//     Term 1 (AT2202-0500)/CC Inputs/Current actual value Ch.9 <-> Data Pointer/CurrentActualValues[8]
//     Term 1 (AT2202-0500)/CC Inputs/Status <-> Data Pointer/Status
//     Term 1 (AT2202-0500)/CC Outputs/Control <-> Data Pointer/Control
//     Term 1 (AT2202-0500)/CC Outputs/Current setpoint value Ch.1 <-> Data Pointer/CurrentSetpointValues[0]
//     Term 1 (AT2202-0500)/CC Outputs/Current setpoint value Ch.10 <-> Data Pointer/CurrentSetpointValues[9]
//     Term 1 (AT2202-0500)/CC Outputs/Current setpoint value Ch.11 <-> Data Pointer/CurrentSetpointValues[10]
//     Term 1 (AT2202-0500)/CC Outputs/Current setpoint value Ch.12 <-> Data Pointer/CurrentSetpointValues[11]
//     Term 1 (AT2202-0500)/CC Outputs/Current setpoint value Ch.13 <-> Data Pointer/CurrentSetpointValues[12]
//     Term 1 (AT2202-0500)/CC Outputs/Current setpoint value Ch.14 <-> Data Pointer/CurrentSetpointValues[13]
//     Term 1 (AT2202-0500)/CC Outputs/Current setpoint value Ch.15 <-> Data Pointer/CurrentSetpointValues[14]
//     Term 1 (AT2202-0500)/CC Outputs/Current setpoint value Ch.16 <-> Data Pointer/CurrentSetpointValues[15]
//     Term 1 (AT2202-0500)/CC Outputs/Current setpoint value Ch.17 <-> Data Pointer/CurrentSetpointValues[16]
//     Term 1 (AT2202-0500)/CC Outputs/Current setpoint value Ch.18 <-> Data Pointer/CurrentSetpointValues[17]
//     Term 1 (AT2202-0500)/CC Outputs/Current setpoint value Ch.19 <-> Data Pointer/CurrentSetpointValues[18]
//     Term 1 (AT2202-0500)/CC Outputs/Current setpoint value Ch.2 <-> Data Pointer/CurrentSetpointValues[1]
//     Term 1 (AT2202-0500)/CC Outputs/Current setpoint value Ch.20 <-> Data Pointer/CurrentSetpointValues[19]
//     Term 1 (AT2202-0500)/CC Outputs/Current setpoint value Ch.21 <-> Data Pointer/CurrentSetpointValues[20]
//     Term 1 (AT2202-0500)/CC Outputs/Current setpoint value Ch.22 <-> Data Pointer/CurrentSetpointValues[21]
//     Term 1 (AT2202-0500)/CC Outputs/Current setpoint value Ch.23 <-> Data Pointer/CurrentSetpointValues[22]
//     Term 1 (AT2202-0500)/CC Outputs/Current setpoint value Ch.24 <-> Data Pointer/CurrentSetpointValues[23]
//     Term 1 (AT2202-0500)/CC Outputs/Current setpoint value Ch.25 <-> Data Pointer/CurrentSetpointValues[24]
//     Term 1 (AT2202-0500)/CC Outputs/Current setpoint value Ch.26 <-> Data Pointer/CurrentSetpointValues[25]
//     Term 1 (AT2202-0500)/CC Outputs/Current setpoint value Ch.27 <-> Data Pointer/CurrentSetpointValues[26]
//     Term 1 (AT2202-0500)/CC Outputs/Current setpoint value Ch.28 <-> Data Pointer/CurrentSetpointValues[27]
//     Term 1 (AT2202-0500)/CC Outputs/Current setpoint value Ch.29 <-> Data Pointer/CurrentSetpointValues[28]
//     Term 1 (AT2202-0500)/CC Outputs/Current setpoint value Ch.3 <-> Data Pointer/CurrentSetpointValues[2]
//     Term 1 (AT2202-0500)/CC Outputs/Current setpoint value Ch.30 <-> Data Pointer/CurrentSetpointValues[29]
//     Term 1 (AT2202-0500)/CC Outputs/Current setpoint value Ch.4 <-> Data Pointer/CurrentSetpointValues[3]
//     Term 1 (AT2202-0500)/CC Outputs/Current setpoint value Ch.5 <-> Data Pointer/CurrentSetpointValues[4]
//     Term 1 (AT2202-0500)/CC Outputs/Current setpoint value Ch.6 <-> Data Pointer/CurrentSetpointValues[5]
//     Term 1 (AT2202-0500)/CC Outputs/Current setpoint value Ch.7 <-> Data Pointer/CurrentSetpointValues[6]
//     Term 1 (AT2202-0500)/CC Outputs/Current setpoint value Ch.8 <-> Data Pointer/CurrentSetpointValues[7]
//     Term 1 (AT2202-0500)/CC Outputs/Current setpoint value Ch.9 <-> Data Pointer/CurrentSetpointValues[8]
//     Term 1 (AT2202-0500)/LFB Inputs/BinaryData <-> Data Pointer/HallSensorValues
//   Device 1 <-> TcCOM Objects/XTS ProcessingUnit 1/Part 1/Module 2
//     Term 2 (AT2200-0500)/CC Inputs/Current actual value Ch.1 <-> Data Pointer/CurrentActualValues[0]
//     Term 2 (AT2200-0500)/CC Inputs/Current actual value Ch.10 <-> Data Pointer/CurrentActualValues[9]
//     Term 2 (AT2200-0500)/CC Inputs/Current actual value Ch.11 <-> Data Pointer/CurrentActualValues[10]
//     Term 2 (AT2200-0500)/CC Inputs/Current actual value Ch.12 <-> Data Pointer/CurrentActualValues[11]
//     Term 2 (AT2200-0500)/CC Inputs/Current actual value Ch.13 <-> Data Pointer/CurrentActualValues[12]
//     Term 2 (AT2200-0500)/CC Inputs/Current actual value Ch.14 <-> Data Pointer/CurrentActualValues[13]
//     Term 2 (AT2200-0500)/CC Inputs/Current actual value Ch.15 <-> Data Pointer/CurrentActualValues[14]
//     Term 2 (AT2200-0500)/CC Inputs/Current actual value Ch.16 <-> Data Pointer/CurrentActualValues[15]
//     Term 2 (AT2200-0500)/CC Inputs/Current actual value Ch.17 <-> Data Pointer/CurrentActualValues[16]
//     Term 2 (AT2200-0500)/CC Inputs/Current actual value Ch.18 <-> Data Pointer/CurrentActualValues[17]
//     Term 2 (AT2200-0500)/CC Inputs/Current actual value Ch.19 <-> Data Pointer/CurrentActualValues[18]
//     Term 2 (AT2200-0500)/CC Inputs/Current actual value Ch.2 <-> Data Pointer/CurrentActualValues[1]
//     Term 2 (AT2200-0500)/CC Inputs/Current actual value Ch.20 <-> Data Pointer/CurrentActualValues[19]
//     Term 2 (AT2200-0500)/CC Inputs/Current actual value Ch.21 <-> Data Pointer/CurrentActualValues[20]
//     Term 2 (AT2200-0500)/CC Inputs/Current actual value Ch.22 <-> Data Pointer/CurrentActualValues[21]
//     Term 2 (AT2200-0500)/CC Inputs/Current actual value Ch.23 <-> Data Pointer/CurrentActualValues[22]
//     Term 2 (AT2200-0500)/CC Inputs/Current actual value Ch.24 <-> Data Pointer/CurrentActualValues[23]
//     Term 2 (AT2200-0500)/CC Inputs/Current actual value Ch.25 <-> Data Pointer/CurrentActualValues[24]
//     Term 2 (AT2200-0500)/CC Inputs/Current actual value Ch.26 <-> Data Pointer/CurrentActualValues[25]
//     Term 2 (AT2200-0500)/CC Inputs/Current actual value Ch.27 <-> Data Pointer/CurrentActualValues[26]
//     Term 2 (AT2200-0500)/CC Inputs/Current actual value Ch.28 <-> Data Pointer/CurrentActualValues[27]
//     Term 2 (AT2200-0500)/CC Inputs/Current actual value Ch.29 <-> Data Pointer/CurrentActualValues[28]
//     Term 2 (AT2200-0500)/CC Inputs/Current actual value Ch.3 <-> Data Pointer/CurrentActualValues[2]
//     Term 2 (AT2200-0500)/CC Inputs/Current actual value Ch.30 <-> Data Pointer/CurrentActualValues[29]
//     Term 2 (AT2200-0500)/CC Inputs/Current actual value Ch.4 <-> Data Pointer/CurrentActualValues[3]
//     Term 2 (AT2200-0500)/CC Inputs/Current actual value Ch.5 <-> Data Pointer/CurrentActualValues[4]
//     Term 2 (AT2200-0500)/CC Inputs/Current actual value Ch.6 <-> Data Pointer/CurrentActualValues[5]
//     Term 2 (AT2200-0500)/CC Inputs/Current actual value Ch.7 <-> Data Pointer/CurrentActualValues[6]
//     Term 2 (AT2200-0500)/CC Inputs/Current actual value Ch.8 <-> Data Pointer/CurrentActualValues[7]
//     Term 2 (AT2200-0500)/CC Inputs/Current actual value Ch.9 <-> Data Pointer/CurrentActualValues[8]
//     Term 2 (AT2200-0500)/CC Inputs/Status <-> Data Pointer/Status
//     Term 2 (AT2200-0500)/CC Outputs/Control <-> Data Pointer/Control
//     Term 2 (AT2200-0500)/CC Outputs/Current setpoint value Ch.1 <-> Data Pointer/CurrentSetpointValues[0]
//     Term 2 (AT2200-0500)/CC Outputs/Current setpoint value Ch.10 <-> Data Pointer/CurrentSetpointValues[9]
//     Term 2 (AT2200-0500)/CC Outputs/Current setpoint value Ch.11 <-> Data Pointer/CurrentSetpointValues[10]
//     Term 2 (AT2200-0500)/CC Outputs/Current setpoint value Ch.12 <-> Data Pointer/CurrentSetpointValues[11]
//     Term 2 (AT2200-0500)/CC Outputs/Current setpoint value Ch.13 <-> Data Pointer/CurrentSetpointValues[12]
//     Term 2 (AT2200-0500)/CC Outputs/Current setpoint value Ch.14 <-> Data Pointer/CurrentSetpointValues[13]
//     Term 2 (AT2200-0500)/CC Outputs/Current setpoint value Ch.15 <-> Data Pointer/CurrentSetpointValues[14]
//     Term 2 (AT2200-0500)/CC Outputs/Current setpoint value Ch.16 <-> Data Pointer/CurrentSetpointValues[15]
//     Term 2 (AT2200-0500)/CC Outputs/Current setpoint value Ch.17 <-> Data Pointer/CurrentSetpointValues[16]
//     Term 2 (AT2200-0500)/CC Outputs/Current setpoint value Ch.18 <-> Data Pointer/CurrentSetpointValues[17]
//     Term 2 (AT2200-0500)/CC Outputs/Current setpoint value Ch.19 <-> Data Pointer/CurrentSetpointValues[18]
//     Term 2 (AT2200-0500)/CC Outputs/Current setpoint value Ch.2 <-> Data Pointer/CurrentSetpointValues[1]
//     Term 2 (AT2200-0500)/CC Outputs/Current setpoint value Ch.20 <-> Data Pointer/CurrentSetpointValues[19]
//     Term 2 (AT2200-0500)/CC Outputs/Current setpoint value Ch.21 <-> Data Pointer/CurrentSetpointValues[20]
//     Term 2 (AT2200-0500)/CC Outputs/Current setpoint value Ch.22 <-> Data Pointer/CurrentSetpointValues[21]
//     Term 2 (AT2200-0500)/CC Outputs/Current setpoint value Ch.23 <-> Data Pointer/CurrentSetpointValues[22]
//     Term 2 (AT2200-0500)/CC Outputs/Current setpoint value Ch.24 <-> Data Pointer/CurrentSetpointValues[23]
//     Term 2 (AT2200-0500)/CC Outputs/Current setpoint value Ch.25 <-> Data Pointer/CurrentSetpointValues[24]
//     Term 2 (AT2200-0500)/CC Outputs/Current setpoint value Ch.26 <-> Data Pointer/CurrentSetpointValues[25]
//     Term 2 (AT2200-0500)/CC Outputs/Current setpoint value Ch.27 <-> Data Pointer/CurrentSetpointValues[26]
//     Term 2 (AT2200-0500)/CC Outputs/Current setpoint value Ch.28 <-> Data Pointer/CurrentSetpointValues[27]
//     Term 2 (AT2200-0500)/CC Outputs/Current setpoint value Ch.29 <-> Data Pointer/CurrentSetpointValues[28]
//     Term 2 (AT2200-0500)/CC Outputs/Current setpoint value Ch.3 <-> Data Pointer/CurrentSetpointValues[2]
//     Term 2 (AT2200-0500)/CC Outputs/Current setpoint value Ch.30 <-> Data Pointer/CurrentSetpointValues[29]
//     Term 2 (AT2200-0500)/CC Outputs/Current setpoint value Ch.4 <-> Data Pointer/CurrentSetpointValues[3]
//     Term 2 (AT2200-0500)/CC Outputs/Current setpoint value Ch.5 <-> Data Pointer/CurrentSetpointValues[4]
//     Term 2 (AT2200-0500)/CC Outputs/Current setpoint value Ch.6 <-> Data Pointer/CurrentSetpointValues[5]
//     Term 2 (AT2200-0500)/CC Outputs/Current setpoint value Ch.7 <-> Data Pointer/CurrentSetpointValues[6]
//     Term 2 (AT2200-0500)/CC Outputs/Current setpoint value Ch.8 <-> Data Pointer/CurrentSetpointValues[7]
//     Term 2 (AT2200-0500)/CC Outputs/Current setpoint value Ch.9 <-> Data Pointer/CurrentSetpointValues[8]
//     Term 2 (AT2200-0500)/LFB Inputs/BinaryData <-> Data Pointer/HallSensorValues
//   Device 1 <-> TcCOM Objects/XTS ProcessingUnit 1/Part 1/Module 3
//     Term 3 (AT2200-0500)/CC Inputs/Current actual value Ch.1 <-> Data Pointer/CurrentActualValues[0]
//     Term 3 (AT2200-0500)/CC Inputs/Current actual value Ch.10 <-> Data Pointer/CurrentActualValues[9]
//     Term 3 (AT2200-0500)/CC Inputs/Current actual value Ch.11 <-> Data Pointer/CurrentActualValues[10]
//     Term 3 (AT2200-0500)/CC Inputs/Current actual value Ch.12 <-> Data Pointer/CurrentActualValues[11]
//     Term 3 (AT2200-0500)/CC Inputs/Current actual value Ch.13 <-> Data Pointer/CurrentActualValues[12]
//     Term 3 (AT2200-0500)/CC Inputs/Current actual value Ch.14 <-> Data Pointer/CurrentActualValues[13]
//     Term 3 (AT2200-0500)/CC Inputs/Current actual value Ch.15 <-> Data Pointer/CurrentActualValues[14]
//     Term 3 (AT2200-0500)/CC Inputs/Current actual value Ch.16 <-> Data Pointer/CurrentActualValues[15]
//     Term 3 (AT2200-0500)/CC Inputs/Current actual value Ch.17 <-> Data Pointer/CurrentActualValues[16]
//     Term 3 (AT2200-0500)/CC Inputs/Current actual value Ch.18 <-> Data Pointer/CurrentActualValues[17]
//     Term 3 (AT2200-0500)/CC Inputs/Current actual value Ch.19 <-> Data Pointer/CurrentActualValues[18]
//     Term 3 (AT2200-0500)/CC Inputs/Current actual value Ch.2 <-> Data Pointer/CurrentActualValues[1]
//     Term 3 (AT2200-0500)/CC Inputs/Current actual value Ch.20 <-> Data Pointer/CurrentActualValues[19]
//     Term 3 (AT2200-0500)/CC Inputs/Current actual value Ch.21 <-> Data Pointer/CurrentActualValues[20]
//     Term 3 (AT2200-0500)/CC Inputs/Current actual value Ch.22 <-> Data Pointer/CurrentActualValues[21]
//     Term 3 (AT2200-0500)/CC Inputs/Current actual value Ch.23 <-> Data Pointer/CurrentActualValues[22]
//     Term 3 (AT2200-0500)/CC Inputs/Current actual value Ch.24 <-> Data Pointer/CurrentActualValues[23]
//     Term 3 (AT2200-0500)/CC Inputs/Current actual value Ch.25 <-> Data Pointer/CurrentActualValues[24]
//     Term 3 (AT2200-0500)/CC Inputs/Current actual value Ch.26 <-> Data Pointer/CurrentActualValues[25]
//     Term 3 (AT2200-0500)/CC Inputs/Current actual value Ch.27 <-> Data Pointer/CurrentActualValues[26]
//     Term 3 (AT2200-0500)/CC Inputs/Current actual value Ch.28 <-> Data Pointer/CurrentActualValues[27]
//     Term 3 (AT2200-0500)/CC Inputs/Current actual value Ch.29 <-> Data Pointer/CurrentActualValues[28]
//     Term 3 (AT2200-0500)/CC Inputs/Current actual value Ch.3 <-> Data Pointer/CurrentActualValues[2]
//     Term 3 (AT2200-0500)/CC Inputs/Current actual value Ch.30 <-> Data Pointer/CurrentActualValues[29]
//     Term 3 (AT2200-0500)/CC Inputs/Current actual value Ch.4 <-> Data Pointer/CurrentActualValues[3]
//     Term 3 (AT2200-0500)/CC Inputs/Current actual value Ch.5 <-> Data Pointer/CurrentActualValues[4]
//     Term 3 (AT2200-0500)/CC Inputs/Current actual value Ch.6 <-> Data Pointer/CurrentActualValues[5]
//     Term 3 (AT2200-0500)/CC Inputs/Current actual value Ch.7 <-> Data Pointer/CurrentActualValues[6]
//     Term 3 (AT2200-0500)/CC Inputs/Current actual value Ch.8 <-> Data Pointer/CurrentActualValues[7]
//     Term 3 (AT2200-0500)/CC Inputs/Current actual value Ch.9 <-> Data Pointer/CurrentActualValues[8]
//     Term 3 (AT2200-0500)/CC Inputs/Status <-> Data Pointer/Status
//     Term 3 (AT2200-0500)/CC Outputs/Control <-> Data Pointer/Control
//     Term 3 (AT2200-0500)/CC Outputs/Current setpoint value Ch.1 <-> Data Pointer/CurrentSetpointValues[0]
//     Term 3 (AT2200-0500)/CC Outputs/Current setpoint value Ch.10 <-> Data Pointer/CurrentSetpointValues[9]
//     Term 3 (AT2200-0500)/CC Outputs/Current setpoint value Ch.11 <-> Data Pointer/CurrentSetpointValues[10]
//     Term 3 (AT2200-0500)/CC Outputs/Current setpoint value Ch.12 <-> Data Pointer/CurrentSetpointValues[11]
//     Term 3 (AT2200-0500)/CC Outputs/Current setpoint value Ch.13 <-> Data Pointer/CurrentSetpointValues[12]
//     Term 3 (AT2200-0500)/CC Outputs/Current setpoint value Ch.14 <-> Data Pointer/CurrentSetpointValues[13]
//     Term 3 (AT2200-0500)/CC Outputs/Current setpoint value Ch.15 <-> Data Pointer/CurrentSetpointValues[14]
//     Term 3 (AT2200-0500)/CC Outputs/Current setpoint value Ch.16 <-> Data Pointer/CurrentSetpointValues[15]
//     Term 3 (AT2200-0500)/CC Outputs/Current setpoint value Ch.17 <-> Data Pointer/CurrentSetpointValues[16]
//     Term 3 (AT2200-0500)/CC Outputs/Current setpoint value Ch.18 <-> Data Pointer/CurrentSetpointValues[17]
//     Term 3 (AT2200-0500)/CC Outputs/Current setpoint value Ch.19 <-> Data Pointer/CurrentSetpointValues[18]
//     Term 3 (AT2200-0500)/CC Outputs/Current setpoint value Ch.2 <-> Data Pointer/CurrentSetpointValues[1]
//     Term 3 (AT2200-0500)/CC Outputs/Current setpoint value Ch.20 <-> Data Pointer/CurrentSetpointValues[19]
//     Term 3 (AT2200-0500)/CC Outputs/Current setpoint value Ch.21 <-> Data Pointer/CurrentSetpointValues[20]
//     Term 3 (AT2200-0500)/CC Outputs/Current setpoint value Ch.22 <-> Data Pointer/CurrentSetpointValues[21]
//     Term 3 (AT2200-0500)/CC Outputs/Current setpoint value Ch.23 <-> Data Pointer/CurrentSetpointValues[22]
//     Term 3 (AT2200-0500)/CC Outputs/Current setpoint value Ch.24 <-> Data Pointer/CurrentSetpointValues[23]
//     Term 3 (AT2200-0500)/CC Outputs/Current setpoint value Ch.25 <-> Data Pointer/CurrentSetpointValues[24]
//     Term 3 (AT2200-0500)/CC Outputs/Current setpoint value Ch.26 <-> Data Pointer/CurrentSetpointValues[25]
//     Term 3 (AT2200-0500)/CC Outputs/Current setpoint value Ch.27 <-> Data Pointer/CurrentSetpointValues[26]
//     Term 3 (AT2200-0500)/CC Outputs/Current setpoint value Ch.28 <-> Data Pointer/CurrentSetpointValues[27]
//     Term 3 (AT2200-0500)/CC Outputs/Current setpoint value Ch.29 <-> Data Pointer/CurrentSetpointValues[28]
//     Term 3 (AT2200-0500)/CC Outputs/Current setpoint value Ch.3 <-> Data Pointer/CurrentSetpointValues[2]
//     Term 3 (AT2200-0500)/CC Outputs/Current setpoint value Ch.30 <-> Data Pointer/CurrentSetpointValues[29]
//     Term 3 (AT2200-0500)/CC Outputs/Current setpoint value Ch.4 <-> Data Pointer/CurrentSetpointValues[3]
//     Term 3 (AT2200-0500)/CC Outputs/Current setpoint value Ch.5 <-> Data Pointer/CurrentSetpointValues[4]
//     Term 3 (AT2200-0500)/CC Outputs/Current setpoint value Ch.6 <-> Data Pointer/CurrentSetpointValues[5]
//     Term 3 (AT2200-0500)/CC Outputs/Current setpoint value Ch.7 <-> Data Pointer/CurrentSetpointValues[6]
//     Term 3 (AT2200-0500)/CC Outputs/Current setpoint value Ch.8 <-> Data Pointer/CurrentSetpointValues[7]
//     Term 3 (AT2200-0500)/CC Outputs/Current setpoint value Ch.9 <-> Data Pointer/CurrentSetpointValues[8]
//     Term 3 (AT2200-0500)/LFB Inputs/BinaryData <-> Data Pointer/HallSensorValues
//   Device 16 <-> TcCOM Objects/XTS ProcessingUnit 1/Part 1/Module 4
//     Term 4 (AT2202-0500)/CC Inputs/Current actual value Ch.1 <-> Data Pointer/CurrentActualValues[0]
//     Term 4 (AT2202-0500)/CC Inputs/Current actual value Ch.10 <-> Data Pointer/CurrentActualValues[9]
//     Term 4 (AT2202-0500)/CC Inputs/Current actual value Ch.11 <-> Data Pointer/CurrentActualValues[10]
//     Term 4 (AT2202-0500)/CC Inputs/Current actual value Ch.12 <-> Data Pointer/CurrentActualValues[11]
//     Term 4 (AT2202-0500)/CC Inputs/Current actual value Ch.13 <-> Data Pointer/CurrentActualValues[12]
//     Term 4 (AT2202-0500)/CC Inputs/Current actual value Ch.14 <-> Data Pointer/CurrentActualValues[13]
//     Term 4 (AT2202-0500)/CC Inputs/Current actual value Ch.15 <-> Data Pointer/CurrentActualValues[14]
//     Term 4 (AT2202-0500)/CC Inputs/Current actual value Ch.16 <-> Data Pointer/CurrentActualValues[15]
//     Term 4 (AT2202-0500)/CC Inputs/Current actual value Ch.17 <-> Data Pointer/CurrentActualValues[16]
//     Term 4 (AT2202-0500)/CC Inputs/Current actual value Ch.18 <-> Data Pointer/CurrentActualValues[17]
//     Term 4 (AT2202-0500)/CC Inputs/Current actual value Ch.19 <-> Data Pointer/CurrentActualValues[18]
//     Term 4 (AT2202-0500)/CC Inputs/Current actual value Ch.2 <-> Data Pointer/CurrentActualValues[1]
//     Term 4 (AT2202-0500)/CC Inputs/Current actual value Ch.20 <-> Data Pointer/CurrentActualValues[19]
//     Term 4 (AT2202-0500)/CC Inputs/Current actual value Ch.21 <-> Data Pointer/CurrentActualValues[20]
//     Term 4 (AT2202-0500)/CC Inputs/Current actual value Ch.22 <-> Data Pointer/CurrentActualValues[21]
//     Term 4 (AT2202-0500)/CC Inputs/Current actual value Ch.23 <-> Data Pointer/CurrentActualValues[22]
//     Term 4 (AT2202-0500)/CC Inputs/Current actual value Ch.24 <-> Data Pointer/CurrentActualValues[23]
//     Term 4 (AT2202-0500)/CC Inputs/Current actual value Ch.25 <-> Data Pointer/CurrentActualValues[24]
//     Term 4 (AT2202-0500)/CC Inputs/Current actual value Ch.26 <-> Data Pointer/CurrentActualValues[25]
//     Term 4 (AT2202-0500)/CC Inputs/Current actual value Ch.27 <-> Data Pointer/CurrentActualValues[26]
//     Term 4 (AT2202-0500)/CC Inputs/Current actual value Ch.28 <-> Data Pointer/CurrentActualValues[27]
//     Term 4 (AT2202-0500)/CC Inputs/Current actual value Ch.29 <-> Data Pointer/CurrentActualValues[28]
//     Term 4 (AT2202-0500)/CC Inputs/Current actual value Ch.3 <-> Data Pointer/CurrentActualValues[2]
//     Term 4 (AT2202-0500)/CC Inputs/Current actual value Ch.30 <-> Data Pointer/CurrentActualValues[29]
//     Term 4 (AT2202-0500)/CC Inputs/Current actual value Ch.4 <-> Data Pointer/CurrentActualValues[3]
//     Term 4 (AT2202-0500)/CC Inputs/Current actual value Ch.5 <-> Data Pointer/CurrentActualValues[4]
//     Term 4 (AT2202-0500)/CC Inputs/Current actual value Ch.6 <-> Data Pointer/CurrentActualValues[5]
//     Term 4 (AT2202-0500)/CC Inputs/Current actual value Ch.7 <-> Data Pointer/CurrentActualValues[6]
//     Term 4 (AT2202-0500)/CC Inputs/Current actual value Ch.8 <-> Data Pointer/CurrentActualValues[7]
//     Term 4 (AT2202-0500)/CC Inputs/Current actual value Ch.9 <-> Data Pointer/CurrentActualValues[8]
//     Term 4 (AT2202-0500)/CC Inputs/Status <-> Data Pointer/Status
//     Term 4 (AT2202-0500)/CC Outputs/Control <-> Data Pointer/Control
//     Term 4 (AT2202-0500)/CC Outputs/Current setpoint value Ch.1 <-> Data Pointer/CurrentSetpointValues[0]
//     Term 4 (AT2202-0500)/CC Outputs/Current setpoint value Ch.10 <-> Data Pointer/CurrentSetpointValues[9]
//     Term 4 (AT2202-0500)/CC Outputs/Current setpoint value Ch.11 <-> Data Pointer/CurrentSetpointValues[10]
//     Term 4 (AT2202-0500)/CC Outputs/Current setpoint value Ch.12 <-> Data Pointer/CurrentSetpointValues[11]
//     Term 4 (AT2202-0500)/CC Outputs/Current setpoint value Ch.13 <-> Data Pointer/CurrentSetpointValues[12]
//     Term 4 (AT2202-0500)/CC Outputs/Current setpoint value Ch.14 <-> Data Pointer/CurrentSetpointValues[13]
//     Term 4 (AT2202-0500)/CC Outputs/Current setpoint value Ch.15 <-> Data Pointer/CurrentSetpointValues[14]
//     Term 4 (AT2202-0500)/CC Outputs/Current setpoint value Ch.16 <-> Data Pointer/CurrentSetpointValues[15]
//     Term 4 (AT2202-0500)/CC Outputs/Current setpoint value Ch.17 <-> Data Pointer/CurrentSetpointValues[16]
//     Term 4 (AT2202-0500)/CC Outputs/Current setpoint value Ch.18 <-> Data Pointer/CurrentSetpointValues[17]
//     Term 4 (AT2202-0500)/CC Outputs/Current setpoint value Ch.19 <-> Data Pointer/CurrentSetpointValues[18]
//     Term 4 (AT2202-0500)/CC Outputs/Current setpoint value Ch.2 <-> Data Pointer/CurrentSetpointValues[1]
//     Term 4 (AT2202-0500)/CC Outputs/Current setpoint value Ch.20 <-> Data Pointer/CurrentSetpointValues[19]
//     Term 4 (AT2202-0500)/CC Outputs/Current setpoint value Ch.21 <-> Data Pointer/CurrentSetpointValues[20]
//     Term 4 (AT2202-0500)/CC Outputs/Current setpoint value Ch.22 <-> Data Pointer/CurrentSetpointValues[21]
//     Term 4 (AT2202-0500)/CC Outputs/Current setpoint value Ch.23 <-> Data Pointer/CurrentSetpointValues[22]
//     Term 4 (AT2202-0500)/CC Outputs/Current setpoint value Ch.24 <-> Data Pointer/CurrentSetpointValues[23]
//     Term 4 (AT2202-0500)/CC Outputs/Current setpoint value Ch.25 <-> Data Pointer/CurrentSetpointValues[24]
//     Term 4 (AT2202-0500)/CC Outputs/Current setpoint value Ch.26 <-> Data Pointer/CurrentSetpointValues[25]
//     Term 4 (AT2202-0500)/CC Outputs/Current setpoint value Ch.27 <-> Data Pointer/CurrentSetpointValues[26]
//     Term 4 (AT2202-0500)/CC Outputs/Current setpoint value Ch.28 <-> Data Pointer/CurrentSetpointValues[27]
//     Term 4 (AT2202-0500)/CC Outputs/Current setpoint value Ch.29 <-> Data Pointer/CurrentSetpointValues[28]
//     Term 4 (AT2202-0500)/CC Outputs/Current setpoint value Ch.3 <-> Data Pointer/CurrentSetpointValues[2]
//     Term 4 (AT2202-0500)/CC Outputs/Current setpoint value Ch.30 <-> Data Pointer/CurrentSetpointValues[29]
//     Term 4 (AT2202-0500)/CC Outputs/Current setpoint value Ch.4 <-> Data Pointer/CurrentSetpointValues[3]
//     Term 4 (AT2202-0500)/CC Outputs/Current setpoint value Ch.5 <-> Data Pointer/CurrentSetpointValues[4]
//     Term 4 (AT2202-0500)/CC Outputs/Current setpoint value Ch.6 <-> Data Pointer/CurrentSetpointValues[5]
//     Term 4 (AT2202-0500)/CC Outputs/Current setpoint value Ch.7 <-> Data Pointer/CurrentSetpointValues[6]
//     Term 4 (AT2202-0500)/CC Outputs/Current setpoint value Ch.8 <-> Data Pointer/CurrentSetpointValues[7]
//     Term 4 (AT2202-0500)/CC Outputs/Current setpoint value Ch.9 <-> Data Pointer/CurrentSetpointValues[8]
//     Term 4 (AT2202-0500)/LFB Inputs/BinaryData <-> Data Pointer/HallSensorValues
//   Device 16 <-> TcCOM Objects/XTS ProcessingUnit 1/Part 1/Module 5
//     Term 5 (AT2200-0500)/CC Inputs/Current actual value Ch.1 <-> Data Pointer/CurrentActualValues[0]
//     Term 5 (AT2200-0500)/CC Inputs/Current actual value Ch.10 <-> Data Pointer/CurrentActualValues[9]
//     Term 5 (AT2200-0500)/CC Inputs/Current actual value Ch.11 <-> Data Pointer/CurrentActualValues[10]
//     Term 5 (AT2200-0500)/CC Inputs/Current actual value Ch.12 <-> Data Pointer/CurrentActualValues[11]
//     Term 5 (AT2200-0500)/CC Inputs/Current actual value Ch.13 <-> Data Pointer/CurrentActualValues[12]
//     Term 5 (AT2200-0500)/CC Inputs/Current actual value Ch.14 <-> Data Pointer/CurrentActualValues[13]
//     Term 5 (AT2200-0500)/CC Inputs/Current actual value Ch.15 <-> Data Pointer/CurrentActualValues[14]
//     Term 5 (AT2200-0500)/CC Inputs/Current actual value Ch.16 <-> Data Pointer/CurrentActualValues[15]
//     Term 5 (AT2200-0500)/CC Inputs/Current actual value Ch.17 <-> Data Pointer/CurrentActualValues[16]
//     Term 5 (AT2200-0500)/CC Inputs/Current actual value Ch.18 <-> Data Pointer/CurrentActualValues[17]
//     Term 5 (AT2200-0500)/CC Inputs/Current actual value Ch.19 <-> Data Pointer/CurrentActualValues[18]
//     Term 5 (AT2200-0500)/CC Inputs/Current actual value Ch.2 <-> Data Pointer/CurrentActualValues[1]
//     Term 5 (AT2200-0500)/CC Inputs/Current actual value Ch.20 <-> Data Pointer/CurrentActualValues[19]
//     Term 5 (AT2200-0500)/CC Inputs/Current actual value Ch.21 <-> Data Pointer/CurrentActualValues[20]
//     Term 5 (AT2200-0500)/CC Inputs/Current actual value Ch.22 <-> Data Pointer/CurrentActualValues[21]
//     Term 5 (AT2200-0500)/CC Inputs/Current actual value Ch.23 <-> Data Pointer/CurrentActualValues[22]
//     Term 5 (AT2200-0500)/CC Inputs/Current actual value Ch.24 <-> Data Pointer/CurrentActualValues[23]
//     Term 5 (AT2200-0500)/CC Inputs/Current actual value Ch.25 <-> Data Pointer/CurrentActualValues[24]
//     Term 5 (AT2200-0500)/CC Inputs/Current actual value Ch.26 <-> Data Pointer/CurrentActualValues[25]
//     Term 5 (AT2200-0500)/CC Inputs/Current actual value Ch.27 <-> Data Pointer/CurrentActualValues[26]
//     Term 5 (AT2200-0500)/CC Inputs/Current actual value Ch.28 <-> Data Pointer/CurrentActualValues[27]
//     Term 5 (AT2200-0500)/CC Inputs/Current actual value Ch.29 <-> Data Pointer/CurrentActualValues[28]
//     Term 5 (AT2200-0500)/CC Inputs/Current actual value Ch.3 <-> Data Pointer/CurrentActualValues[2]
//     Term 5 (AT2200-0500)/CC Inputs/Current actual value Ch.30 <-> Data Pointer/CurrentActualValues[29]
//     Term 5 (AT2200-0500)/CC Inputs/Current actual value Ch.4 <-> Data Pointer/CurrentActualValues[3]
//     Term 5 (AT2200-0500)/CC Inputs/Current actual value Ch.5 <-> Data Pointer/CurrentActualValues[4]
//     Term 5 (AT2200-0500)/CC Inputs/Current actual value Ch.6 <-> Data Pointer/CurrentActualValues[5]
//     Term 5 (AT2200-0500)/CC Inputs/Current actual value Ch.7 <-> Data Pointer/CurrentActualValues[6]
//     Term 5 (AT2200-0500)/CC Inputs/Current actual value Ch.8 <-> Data Pointer/CurrentActualValues[7]
//     Term 5 (AT2200-0500)/CC Inputs/Current actual value Ch.9 <-> Data Pointer/CurrentActualValues[8]
//     Term 5 (AT2200-0500)/CC Inputs/Status <-> Data Pointer/Status
//     Term 5 (AT2200-0500)/CC Outputs/Control <-> Data Pointer/Control
//     Term 5 (AT2200-0500)/CC Outputs/Current setpoint value Ch.1 <-> Data Pointer/CurrentSetpointValues[0]
//     Term 5 (AT2200-0500)/CC Outputs/Current setpoint value Ch.10 <-> Data Pointer/CurrentSetpointValues[9]
//     Term 5 (AT2200-0500)/CC Outputs/Current setpoint value Ch.11 <-> Data Pointer/CurrentSetpointValues[10]
//     Term 5 (AT2200-0500)/CC Outputs/Current setpoint value Ch.12 <-> Data Pointer/CurrentSetpointValues[11]
//     Term 5 (AT2200-0500)/CC Outputs/Current setpoint value Ch.13 <-> Data Pointer/CurrentSetpointValues[12]
//     Term 5 (AT2200-0500)/CC Outputs/Current setpoint value Ch.14 <-> Data Pointer/CurrentSetpointValues[13]
//     Term 5 (AT2200-0500)/CC Outputs/Current setpoint value Ch.15 <-> Data Pointer/CurrentSetpointValues[14]
//     Term 5 (AT2200-0500)/CC Outputs/Current setpoint value Ch.16 <-> Data Pointer/CurrentSetpointValues[15]
//     Term 5 (AT2200-0500)/CC Outputs/Current setpoint value Ch.17 <-> Data Pointer/CurrentSetpointValues[16]
//     Term 5 (AT2200-0500)/CC Outputs/Current setpoint value Ch.18 <-> Data Pointer/CurrentSetpointValues[17]
//     Term 5 (AT2200-0500)/CC Outputs/Current setpoint value Ch.19 <-> Data Pointer/CurrentSetpointValues[18]
//     Term 5 (AT2200-0500)/CC Outputs/Current setpoint value Ch.2 <-> Data Pointer/CurrentSetpointValues[1]
//     Term 5 (AT2200-0500)/CC Outputs/Current setpoint value Ch.20 <-> Data Pointer/CurrentSetpointValues[19]
//     Term 5 (AT2200-0500)/CC Outputs/Current setpoint value Ch.21 <-> Data Pointer/CurrentSetpointValues[20]
//     Term 5 (AT2200-0500)/CC Outputs/Current setpoint value Ch.22 <-> Data Pointer/CurrentSetpointValues[21]
//     Term 5 (AT2200-0500)/CC Outputs/Current setpoint value Ch.23 <-> Data Pointer/CurrentSetpointValues[22]
//     Term 5 (AT2200-0500)/CC Outputs/Current setpoint value Ch.24 <-> Data Pointer/CurrentSetpointValues[23]
//     Term 5 (AT2200-0500)/CC Outputs/Current setpoint value Ch.25 <-> Data Pointer/CurrentSetpointValues[24]
//     Term 5 (AT2200-0500)/CC Outputs/Current setpoint value Ch.26 <-> Data Pointer/CurrentSetpointValues[25]
//     Term 5 (AT2200-0500)/CC Outputs/Current setpoint value Ch.27 <-> Data Pointer/CurrentSetpointValues[26]
//     Term 5 (AT2200-0500)/CC Outputs/Current setpoint value Ch.28 <-> Data Pointer/CurrentSetpointValues[27]
//     Term 5 (AT2200-0500)/CC Outputs/Current setpoint value Ch.29 <-> Data Pointer/CurrentSetpointValues[28]
//     Term 5 (AT2200-0500)/CC Outputs/Current setpoint value Ch.3 <-> Data Pointer/CurrentSetpointValues[2]
//     Term 5 (AT2200-0500)/CC Outputs/Current setpoint value Ch.30 <-> Data Pointer/CurrentSetpointValues[29]
//     Term 5 (AT2200-0500)/CC Outputs/Current setpoint value Ch.4 <-> Data Pointer/CurrentSetpointValues[3]
//     Term 5 (AT2200-0500)/CC Outputs/Current setpoint value Ch.5 <-> Data Pointer/CurrentSetpointValues[4]
//     Term 5 (AT2200-0500)/CC Outputs/Current setpoint value Ch.6 <-> Data Pointer/CurrentSetpointValues[5]
//     Term 5 (AT2200-0500)/CC Outputs/Current setpoint value Ch.7 <-> Data Pointer/CurrentSetpointValues[6]
//     Term 5 (AT2200-0500)/CC Outputs/Current setpoint value Ch.8 <-> Data Pointer/CurrentSetpointValues[7]
//     Term 5 (AT2200-0500)/CC Outputs/Current setpoint value Ch.9 <-> Data Pointer/CurrentSetpointValues[8]
//     Term 5 (AT2200-0500)/LFB Inputs/BinaryData <-> Data Pointer/HallSensorValues
//   Device 16 <-> TcCOM Objects/XTS ProcessingUnit 1/Part 1/Module 6
//     Term 6 (AT2200-0500)/CC Inputs/Current actual value Ch.1 <-> Data Pointer/CurrentActualValues[0]
//     Term 6 (AT2200-0500)/CC Inputs/Current actual value Ch.10 <-> Data Pointer/CurrentActualValues[9]
//     Term 6 (AT2200-0500)/CC Inputs/Current actual value Ch.11 <-> Data Pointer/CurrentActualValues[10]
//     Term 6 (AT2200-0500)/CC Inputs/Current actual value Ch.12 <-> Data Pointer/CurrentActualValues[11]
//     Term 6 (AT2200-0500)/CC Inputs/Current actual value Ch.13 <-> Data Pointer/CurrentActualValues[12]
//     Term 6 (AT2200-0500)/CC Inputs/Current actual value Ch.14 <-> Data Pointer/CurrentActualValues[13]
//     Term 6 (AT2200-0500)/CC Inputs/Current actual value Ch.15 <-> Data Pointer/CurrentActualValues[14]
//     Term 6 (AT2200-0500)/CC Inputs/Current actual value Ch.16 <-> Data Pointer/CurrentActualValues[15]
//     Term 6 (AT2200-0500)/CC Inputs/Current actual value Ch.17 <-> Data Pointer/CurrentActualValues[16]
//     Term 6 (AT2200-0500)/CC Inputs/Current actual value Ch.18 <-> Data Pointer/CurrentActualValues[17]
//     Term 6 (AT2200-0500)/CC Inputs/Current actual value Ch.19 <-> Data Pointer/CurrentActualValues[18]
//     Term 6 (AT2200-0500)/CC Inputs/Current actual value Ch.2 <-> Data Pointer/CurrentActualValues[1]
//     Term 6 (AT2200-0500)/CC Inputs/Current actual value Ch.20 <-> Data Pointer/CurrentActualValues[19]
//     Term 6 (AT2200-0500)/CC Inputs/Current actual value Ch.21 <-> Data Pointer/CurrentActualValues[20]
//     Term 6 (AT2200-0500)/CC Inputs/Current actual value Ch.22 <-> Data Pointer/CurrentActualValues[21]
//     Term 6 (AT2200-0500)/CC Inputs/Current actual value Ch.23 <-> Data Pointer/CurrentActualValues[22]
//     Term 6 (AT2200-0500)/CC Inputs/Current actual value Ch.24 <-> Data Pointer/CurrentActualValues[23]
//     Term 6 (AT2200-0500)/CC Inputs/Current actual value Ch.25 <-> Data Pointer/CurrentActualValues[24]
//     Term 6 (AT2200-0500)/CC Inputs/Current actual value Ch.26 <-> Data Pointer/CurrentActualValues[25]
//     Term 6 (AT2200-0500)/CC Inputs/Current actual value Ch.27 <-> Data Pointer/CurrentActualValues[26]
//     Term 6 (AT2200-0500)/CC Inputs/Current actual value Ch.28 <-> Data Pointer/CurrentActualValues[27]
//     Term 6 (AT2200-0500)/CC Inputs/Current actual value Ch.29 <-> Data Pointer/CurrentActualValues[28]
//     Term 6 (AT2200-0500)/CC Inputs/Current actual value Ch.3 <-> Data Pointer/CurrentActualValues[2]
//     Term 6 (AT2200-0500)/CC Inputs/Current actual value Ch.30 <-> Data Pointer/CurrentActualValues[29]
//     Term 6 (AT2200-0500)/CC Inputs/Current actual value Ch.4 <-> Data Pointer/CurrentActualValues[3]
//     Term 6 (AT2200-0500)/CC Inputs/Current actual value Ch.5 <-> Data Pointer/CurrentActualValues[4]
//     Term 6 (AT2200-0500)/CC Inputs/Current actual value Ch.6 <-> Data Pointer/CurrentActualValues[5]
//     Term 6 (AT2200-0500)/CC Inputs/Current actual value Ch.7 <-> Data Pointer/CurrentActualValues[6]
//     Term 6 (AT2200-0500)/CC Inputs/Current actual value Ch.8 <-> Data Pointer/CurrentActualValues[7]
//     Term 6 (AT2200-0500)/CC Inputs/Current actual value Ch.9 <-> Data Pointer/CurrentActualValues[8]
//     Term 6 (AT2200-0500)/CC Inputs/Status <-> Data Pointer/Status
//     Term 6 (AT2200-0500)/CC Outputs/Control <-> Data Pointer/Control
//     Term 6 (AT2200-0500)/CC Outputs/Current setpoint value Ch.1 <-> Data Pointer/CurrentSetpointValues[0]
//     Term 6 (AT2200-0500)/CC Outputs/Current setpoint value Ch.10 <-> Data Pointer/CurrentSetpointValues[9]
//     Term 6 (AT2200-0500)/CC Outputs/Current setpoint value Ch.11 <-> Data Pointer/CurrentSetpointValues[10]
//     Term 6 (AT2200-0500)/CC Outputs/Current setpoint value Ch.12 <-> Data Pointer/CurrentSetpointValues[11]
//     Term 6 (AT2200-0500)/CC Outputs/Current setpoint value Ch.13 <-> Data Pointer/CurrentSetpointValues[12]
//     Term 6 (AT2200-0500)/CC Outputs/Current setpoint value Ch.14 <-> Data Pointer/CurrentSetpointValues[13]
//     Term 6 (AT2200-0500)/CC Outputs/Current setpoint value Ch.15 <-> Data Pointer/CurrentSetpointValues[14]
//     Term 6 (AT2200-0500)/CC Outputs/Current setpoint value Ch.16 <-> Data Pointer/CurrentSetpointValues[15]
//     Term 6 (AT2200-0500)/CC Outputs/Current setpoint value Ch.17 <-> Data Pointer/CurrentSetpointValues[16]
//     Term 6 (AT2200-0500)/CC Outputs/Current setpoint value Ch.18 <-> Data Pointer/CurrentSetpointValues[17]
//     Term 6 (AT2200-0500)/CC Outputs/Current setpoint value Ch.19 <-> Data Pointer/CurrentSetpointValues[18]
//     Term 6 (AT2200-0500)/CC Outputs/Current setpoint value Ch.2 <-> Data Pointer/CurrentSetpointValues[1]
//     Term 6 (AT2200-0500)/CC Outputs/Current setpoint value Ch.20 <-> Data Pointer/CurrentSetpointValues[19]
//     Term 6 (AT2200-0500)/CC Outputs/Current setpoint value Ch.21 <-> Data Pointer/CurrentSetpointValues[20]
//     Term 6 (AT2200-0500)/CC Outputs/Current setpoint value Ch.22 <-> Data Pointer/CurrentSetpointValues[21]
//     Term 6 (AT2200-0500)/CC Outputs/Current setpoint value Ch.23 <-> Data Pointer/CurrentSetpointValues[22]
//     Term 6 (AT2200-0500)/CC Outputs/Current setpoint value Ch.24 <-> Data Pointer/CurrentSetpointValues[23]
//     Term 6 (AT2200-0500)/CC Outputs/Current setpoint value Ch.25 <-> Data Pointer/CurrentSetpointValues[24]
//     Term 6 (AT2200-0500)/CC Outputs/Current setpoint value Ch.26 <-> Data Pointer/CurrentSetpointValues[25]
//     Term 6 (AT2200-0500)/CC Outputs/Current setpoint value Ch.27 <-> Data Pointer/CurrentSetpointValues[26]
//     Term 6 (AT2200-0500)/CC Outputs/Current setpoint value Ch.28 <-> Data Pointer/CurrentSetpointValues[27]
//     Term 6 (AT2200-0500)/CC Outputs/Current setpoint value Ch.29 <-> Data Pointer/CurrentSetpointValues[28]
//     Term 6 (AT2200-0500)/CC Outputs/Current setpoint value Ch.3 <-> Data Pointer/CurrentSetpointValues[2]
//     Term 6 (AT2200-0500)/CC Outputs/Current setpoint value Ch.30 <-> Data Pointer/CurrentSetpointValues[29]
//     Term 6 (AT2200-0500)/CC Outputs/Current setpoint value Ch.4 <-> Data Pointer/CurrentSetpointValues[3]
//     Term 6 (AT2200-0500)/CC Outputs/Current setpoint value Ch.5 <-> Data Pointer/CurrentSetpointValues[4]
//     Term 6 (AT2200-0500)/CC Outputs/Current setpoint value Ch.6 <-> Data Pointer/CurrentSetpointValues[5]
//     Term 6 (AT2200-0500)/CC Outputs/Current setpoint value Ch.7 <-> Data Pointer/CurrentSetpointValues[6]
//     Term 6 (AT2200-0500)/CC Outputs/Current setpoint value Ch.8 <-> Data Pointer/CurrentSetpointValues[7]
//     Term 6 (AT2200-0500)/CC Outputs/Current setpoint value Ch.9 <-> Data Pointer/CurrentSetpointValues[8]
//     Term 6 (AT2200-0500)/LFB Inputs/BinaryData <-> Data Pointer/HallSensorValues
//   Device 18 <-> TcCOM Objects/XTS ProcessingUnit 1/Part 1/Module 10
//     Term 11 (AT2040-0250)/CC Inputs/Current actual value Ch.1 <-> Data Pointer/CurrentActualValues[0]
//     Term 11 (AT2040-0250)/CC Inputs/Current actual value Ch.10 <-> Data Pointer/CurrentActualValues[9]
//     Term 11 (AT2040-0250)/CC Inputs/Current actual value Ch.11 <-> Data Pointer/CurrentActualValues[10]
//     Term 11 (AT2040-0250)/CC Inputs/Current actual value Ch.12 <-> Data Pointer/CurrentActualValues[11]
//     Term 11 (AT2040-0250)/CC Inputs/Current actual value Ch.13 <-> Data Pointer/CurrentActualValues[12]
//     Term 11 (AT2040-0250)/CC Inputs/Current actual value Ch.14 <-> Data Pointer/CurrentActualValues[13]
//     Term 11 (AT2040-0250)/CC Inputs/Current actual value Ch.15 <-> Data Pointer/CurrentActualValues[14]
//     Term 11 (AT2040-0250)/CC Inputs/Current actual value Ch.2 <-> Data Pointer/CurrentActualValues[1]
//     Term 11 (AT2040-0250)/CC Inputs/Current actual value Ch.3 <-> Data Pointer/CurrentActualValues[2]
//     Term 11 (AT2040-0250)/CC Inputs/Current actual value Ch.4 <-> Data Pointer/CurrentActualValues[3]
//     Term 11 (AT2040-0250)/CC Inputs/Current actual value Ch.5 <-> Data Pointer/CurrentActualValues[4]
//     Term 11 (AT2040-0250)/CC Inputs/Current actual value Ch.6 <-> Data Pointer/CurrentActualValues[5]
//     Term 11 (AT2040-0250)/CC Inputs/Current actual value Ch.7 <-> Data Pointer/CurrentActualValues[6]
//     Term 11 (AT2040-0250)/CC Inputs/Current actual value Ch.8 <-> Data Pointer/CurrentActualValues[7]
//     Term 11 (AT2040-0250)/CC Inputs/Current actual value Ch.9 <-> Data Pointer/CurrentActualValues[8]
//     Term 11 (AT2040-0250)/CC Inputs/Status <-> Data Pointer/Status
//     Term 11 (AT2040-0250)/CC Outputs/Control <-> Data Pointer/Control
//     Term 11 (AT2040-0250)/CC Outputs/Current setpoint value Ch.1 <-> Data Pointer/CurrentSetpointValues[0]
//     Term 11 (AT2040-0250)/CC Outputs/Current setpoint value Ch.10 <-> Data Pointer/CurrentSetpointValues[9]
//     Term 11 (AT2040-0250)/CC Outputs/Current setpoint value Ch.11 <-> Data Pointer/CurrentSetpointValues[10]
//     Term 11 (AT2040-0250)/CC Outputs/Current setpoint value Ch.12 <-> Data Pointer/CurrentSetpointValues[11]
//     Term 11 (AT2040-0250)/CC Outputs/Current setpoint value Ch.13 <-> Data Pointer/CurrentSetpointValues[12]
//     Term 11 (AT2040-0250)/CC Outputs/Current setpoint value Ch.14 <-> Data Pointer/CurrentSetpointValues[13]
//     Term 11 (AT2040-0250)/CC Outputs/Current setpoint value Ch.15 <-> Data Pointer/CurrentSetpointValues[14]
//     Term 11 (AT2040-0250)/CC Outputs/Current setpoint value Ch.2 <-> Data Pointer/CurrentSetpointValues[1]
//     Term 11 (AT2040-0250)/CC Outputs/Current setpoint value Ch.3 <-> Data Pointer/CurrentSetpointValues[2]
//     Term 11 (AT2040-0250)/CC Outputs/Current setpoint value Ch.4 <-> Data Pointer/CurrentSetpointValues[3]
//     Term 11 (AT2040-0250)/CC Outputs/Current setpoint value Ch.5 <-> Data Pointer/CurrentSetpointValues[4]
//     Term 11 (AT2040-0250)/CC Outputs/Current setpoint value Ch.6 <-> Data Pointer/CurrentSetpointValues[5]
//     Term 11 (AT2040-0250)/CC Outputs/Current setpoint value Ch.7 <-> Data Pointer/CurrentSetpointValues[6]
//     Term 11 (AT2040-0250)/CC Outputs/Current setpoint value Ch.8 <-> Data Pointer/CurrentSetpointValues[7]
//     Term 11 (AT2040-0250)/CC Outputs/Current setpoint value Ch.9 <-> Data Pointer/CurrentSetpointValues[8]
//     Term 11 (AT2040-0250)/Term 12 (AT2040-5250)/FB Inputs/Value Channel 01 <-> Data Pointer/RawPositionValues[0]
//     Term 11 (AT2040-0250)/Term 12 (AT2040-5250)/FB Inputs/Value Channel 02 <-> Data Pointer/RawPositionValues[1]
//     Term 11 (AT2040-0250)/Term 12 (AT2040-5250)/FB Inputs/Value Channel 03 <-> Data Pointer/RawPositionValues[2]
//     Term 11 (AT2040-0250)/Term 12 (AT2040-5250)/FB Inputs/Value Channel 04 <-> Data Pointer/RawPositionValues[3]
//     Term 11 (AT2040-0250)/Term 12 (AT2040-5250)/FB Inputs/Value Channel 05 <-> Data Pointer/RawPositionValues[4]
//     Term 11 (AT2040-0250)/Term 12 (AT2040-5250)/FB Inputs/Value Channel 06 <-> Data Pointer/RawPositionValues[5]
//     Term 11 (AT2040-0250)/Term 12 (AT2040-5250)/FB Inputs/Value Channel 07 <-> Data Pointer/RawPositionValues[6]
//     Term 11 (AT2040-0250)/Term 12 (AT2040-5250)/FB Inputs/Value Channel 08 <-> Data Pointer/RawPositionValues[7]
//     Term 11 (AT2040-0250)/Term 12 (AT2040-5250)/FB Inputs/Value Channel 09 <-> Data Pointer/RawPositionValues[8]
//     Term 11 (AT2040-0250)/Term 12 (AT2040-5250)/FB Inputs/Value Channel 10 <-> Data Pointer/RawPositionValues[9]
//     Term 11 (AT2040-0250)/Term 12 (AT2040-5250)/FB Inputs/Value Channel 11 <-> Data Pointer/RawPositionValues[10]
//     Term 11 (AT2040-0250)/Term 12 (AT2040-5250)/FB Inputs/Value Channel 12 <-> Data Pointer/RawPositionValues[11]
//     Term 11 (AT2040-0250)/Term 12 (AT2040-5250)/FB Inputs/Value Channel 13 <-> Data Pointer/RawPositionValues[12]
//     Term 11 (AT2040-0250)/Term 12 (AT2040-5250)/FB Inputs/Value Channel 14 <-> Data Pointer/RawPositionValues[13]
//     Term 11 (AT2040-0250)/Term 12 (AT2040-5250)/FB Inputs/Value Channel 15 <-> Data Pointer/RawPositionValues[14]
//     Term 11 (AT2040-0250)/Term 12 (AT2040-5250)/FB Inputs/Value Channel 16 <-> Data Pointer/RawPositionValues[15]
//     Term 11 (AT2040-0250)/Term 12 (AT2040-5250)/FB Inputs/Value Channel 17 <-> Data Pointer/RawPositionValues[16]
//     Term 11 (AT2040-0250)/Term 12 (AT2040-5250)/FB Inputs/Value Channel 18 <-> Data Pointer/RawPositionValues[17]
//     Term 11 (AT2040-0250)/Term 12 (AT2040-5250)/FB Inputs/Value Channel 19 <-> Data Pointer/RawPositionValues[18]
//     Term 11 (AT2040-0250)/Term 12 (AT2040-5250)/FB Inputs/Value Channel 20 <-> Data Pointer/RawPositionValues[19]
//     Term 11 (AT2040-0250)/Term 12 (AT2040-5250)/FB Inputs/Value Channel 21 <-> Data Pointer/RawPositionValues[20]
//     Term 11 (AT2040-0250)/Term 12 (AT2040-5250)/FB Inputs/Value Channel 22 <-> Data Pointer/RawPositionValues[21]
//     Term 11 (AT2040-0250)/Term 12 (AT2040-5250)/FB Inputs/Value Channel 23 <-> Data Pointer/RawPositionValues[22]
//     Term 11 (AT2040-0250)/Term 12 (AT2040-5250)/FB Inputs/Value Channel 24 <-> Data Pointer/RawPositionValues[23]
//     Term 11 (AT2040-0250)/Term 12 (AT2040-5250)/FB Inputs/Value Channel 25 <-> Data Pointer/RawPositionValues[24]
//     Term 11 (AT2040-0250)/Term 12 (AT2040-5250)/FB Inputs/Value Channel 26 <-> Data Pointer/RawPositionValues[25]
//     Term 11 (AT2040-0250)/Term 12 (AT2040-5250)/FB Inputs/Value Channel 27 <-> Data Pointer/RawPositionValues[26]
//     Term 11 (AT2040-0250)/Term 12 (AT2040-5250)/FB Inputs/Value Channel 28 <-> Data Pointer/RawPositionValues[27]
//     Term 11 (AT2040-0250)/Term 12 (AT2040-5250)/FB Inputs/Value Channel 29 <-> Data Pointer/RawPositionValues[28]
//     Term 11 (AT2040-0250)/Term 12 (AT2040-5250)/FB Inputs/Value Channel 30 <-> Data Pointer/RawPositionValues[29]
//     Term 11 (AT2040-0250)/Term 12 (AT2040-5250)/FB Inputs/Value Channel 31 <-> Data Pointer/RawPositionValues[30]
//     Term 11 (AT2040-0250)/Term 12 (AT2040-5250)/FB Inputs/Value Channel 32 <-> Data Pointer/RawPositionValues[31]
//   Device 18 <-> TcCOM Objects/XTS ProcessingUnit 1/Part 1/Module 7
//     Term 7 (AT2202-0500)/CC Inputs/Current actual value Ch.1 <-> Data Pointer/CurrentActualValues[0]
//     Term 7 (AT2202-0500)/CC Inputs/Current actual value Ch.10 <-> Data Pointer/CurrentActualValues[9]
//     Term 7 (AT2202-0500)/CC Inputs/Current actual value Ch.11 <-> Data Pointer/CurrentActualValues[10]
//     Term 7 (AT2202-0500)/CC Inputs/Current actual value Ch.12 <-> Data Pointer/CurrentActualValues[11]
//     Term 7 (AT2202-0500)/CC Inputs/Current actual value Ch.13 <-> Data Pointer/CurrentActualValues[12]
//     Term 7 (AT2202-0500)/CC Inputs/Current actual value Ch.14 <-> Data Pointer/CurrentActualValues[13]
//     Term 7 (AT2202-0500)/CC Inputs/Current actual value Ch.15 <-> Data Pointer/CurrentActualValues[14]
//     Term 7 (AT2202-0500)/CC Inputs/Current actual value Ch.16 <-> Data Pointer/CurrentActualValues[15]
//     Term 7 (AT2202-0500)/CC Inputs/Current actual value Ch.17 <-> Data Pointer/CurrentActualValues[16]
//     Term 7 (AT2202-0500)/CC Inputs/Current actual value Ch.18 <-> Data Pointer/CurrentActualValues[17]
//     Term 7 (AT2202-0500)/CC Inputs/Current actual value Ch.19 <-> Data Pointer/CurrentActualValues[18]
//     Term 7 (AT2202-0500)/CC Inputs/Current actual value Ch.2 <-> Data Pointer/CurrentActualValues[1]
//     Term 7 (AT2202-0500)/CC Inputs/Current actual value Ch.20 <-> Data Pointer/CurrentActualValues[19]
//     Term 7 (AT2202-0500)/CC Inputs/Current actual value Ch.21 <-> Data Pointer/CurrentActualValues[20]
//     Term 7 (AT2202-0500)/CC Inputs/Current actual value Ch.22 <-> Data Pointer/CurrentActualValues[21]
//     Term 7 (AT2202-0500)/CC Inputs/Current actual value Ch.23 <-> Data Pointer/CurrentActualValues[22]
//     Term 7 (AT2202-0500)/CC Inputs/Current actual value Ch.24 <-> Data Pointer/CurrentActualValues[23]
//     Term 7 (AT2202-0500)/CC Inputs/Current actual value Ch.25 <-> Data Pointer/CurrentActualValues[24]
//     Term 7 (AT2202-0500)/CC Inputs/Current actual value Ch.26 <-> Data Pointer/CurrentActualValues[25]
//     Term 7 (AT2202-0500)/CC Inputs/Current actual value Ch.27 <-> Data Pointer/CurrentActualValues[26]
//     Term 7 (AT2202-0500)/CC Inputs/Current actual value Ch.28 <-> Data Pointer/CurrentActualValues[27]
//     Term 7 (AT2202-0500)/CC Inputs/Current actual value Ch.29 <-> Data Pointer/CurrentActualValues[28]
//     Term 7 (AT2202-0500)/CC Inputs/Current actual value Ch.3 <-> Data Pointer/CurrentActualValues[2]
//     Term 7 (AT2202-0500)/CC Inputs/Current actual value Ch.30 <-> Data Pointer/CurrentActualValues[29]
//     Term 7 (AT2202-0500)/CC Inputs/Current actual value Ch.4 <-> Data Pointer/CurrentActualValues[3]
//     Term 7 (AT2202-0500)/CC Inputs/Current actual value Ch.5 <-> Data Pointer/CurrentActualValues[4]
//     Term 7 (AT2202-0500)/CC Inputs/Current actual value Ch.6 <-> Data Pointer/CurrentActualValues[5]
//     Term 7 (AT2202-0500)/CC Inputs/Current actual value Ch.7 <-> Data Pointer/CurrentActualValues[6]
//     Term 7 (AT2202-0500)/CC Inputs/Current actual value Ch.8 <-> Data Pointer/CurrentActualValues[7]
//     Term 7 (AT2202-0500)/CC Inputs/Current actual value Ch.9 <-> Data Pointer/CurrentActualValues[8]
//     Term 7 (AT2202-0500)/CC Inputs/Status <-> Data Pointer/Status
//     Term 7 (AT2202-0500)/CC Outputs/Control <-> Data Pointer/Control
//     Term 7 (AT2202-0500)/CC Outputs/Current setpoint value Ch.1 <-> Data Pointer/CurrentSetpointValues[0]
//     Term 7 (AT2202-0500)/CC Outputs/Current setpoint value Ch.10 <-> Data Pointer/CurrentSetpointValues[9]
//     Term 7 (AT2202-0500)/CC Outputs/Current setpoint value Ch.11 <-> Data Pointer/CurrentSetpointValues[10]
//     Term 7 (AT2202-0500)/CC Outputs/Current setpoint value Ch.12 <-> Data Pointer/CurrentSetpointValues[11]
//     Term 7 (AT2202-0500)/CC Outputs/Current setpoint value Ch.13 <-> Data Pointer/CurrentSetpointValues[12]
//     Term 7 (AT2202-0500)/CC Outputs/Current setpoint value Ch.14 <-> Data Pointer/CurrentSetpointValues[13]
//     Term 7 (AT2202-0500)/CC Outputs/Current setpoint value Ch.15 <-> Data Pointer/CurrentSetpointValues[14]
//     Term 7 (AT2202-0500)/CC Outputs/Current setpoint value Ch.16 <-> Data Pointer/CurrentSetpointValues[15]
//     Term 7 (AT2202-0500)/CC Outputs/Current setpoint value Ch.17 <-> Data Pointer/CurrentSetpointValues[16]
//     Term 7 (AT2202-0500)/CC Outputs/Current setpoint value Ch.18 <-> Data Pointer/CurrentSetpointValues[17]
//     Term 7 (AT2202-0500)/CC Outputs/Current setpoint value Ch.19 <-> Data Pointer/CurrentSetpointValues[18]
//     Term 7 (AT2202-0500)/CC Outputs/Current setpoint value Ch.2 <-> Data Pointer/CurrentSetpointValues[1]
//     Term 7 (AT2202-0500)/CC Outputs/Current setpoint value Ch.20 <-> Data Pointer/CurrentSetpointValues[19]
//     Term 7 (AT2202-0500)/CC Outputs/Current setpoint value Ch.21 <-> Data Pointer/CurrentSetpointValues[20]
//     Term 7 (AT2202-0500)/CC Outputs/Current setpoint value Ch.22 <-> Data Pointer/CurrentSetpointValues[21]
//     Term 7 (AT2202-0500)/CC Outputs/Current setpoint value Ch.23 <-> Data Pointer/CurrentSetpointValues[22]
//     Term 7 (AT2202-0500)/CC Outputs/Current setpoint value Ch.24 <-> Data Pointer/CurrentSetpointValues[23]
//     Term 7 (AT2202-0500)/CC Outputs/Current setpoint value Ch.25 <-> Data Pointer/CurrentSetpointValues[24]
//     Term 7 (AT2202-0500)/CC Outputs/Current setpoint value Ch.26 <-> Data Pointer/CurrentSetpointValues[25]
//     Term 7 (AT2202-0500)/CC Outputs/Current setpoint value Ch.27 <-> Data Pointer/CurrentSetpointValues[26]
//     Term 7 (AT2202-0500)/CC Outputs/Current setpoint value Ch.28 <-> Data Pointer/CurrentSetpointValues[27]
//     Term 7 (AT2202-0500)/CC Outputs/Current setpoint value Ch.29 <-> Data Pointer/CurrentSetpointValues[28]
//     Term 7 (AT2202-0500)/CC Outputs/Current setpoint value Ch.3 <-> Data Pointer/CurrentSetpointValues[2]
//     Term 7 (AT2202-0500)/CC Outputs/Current setpoint value Ch.30 <-> Data Pointer/CurrentSetpointValues[29]
//     Term 7 (AT2202-0500)/CC Outputs/Current setpoint value Ch.4 <-> Data Pointer/CurrentSetpointValues[3]
//     Term 7 (AT2202-0500)/CC Outputs/Current setpoint value Ch.5 <-> Data Pointer/CurrentSetpointValues[4]
//     Term 7 (AT2202-0500)/CC Outputs/Current setpoint value Ch.6 <-> Data Pointer/CurrentSetpointValues[5]
//     Term 7 (AT2202-0500)/CC Outputs/Current setpoint value Ch.7 <-> Data Pointer/CurrentSetpointValues[6]
//     Term 7 (AT2202-0500)/CC Outputs/Current setpoint value Ch.8 <-> Data Pointer/CurrentSetpointValues[7]
//     Term 7 (AT2202-0500)/CC Outputs/Current setpoint value Ch.9 <-> Data Pointer/CurrentSetpointValues[8]
//     Term 7 (AT2202-0500)/LFB Inputs/BinaryData <-> Data Pointer/HallSensorValues
//   Device 18 <-> TcCOM Objects/XTS ProcessingUnit 1/Part 1/Module 8
//     Term 8 (AT2200-0500)/CC Inputs/Current actual value Ch.1 <-> Data Pointer/CurrentActualValues[0]
//     Term 8 (AT2200-0500)/CC Inputs/Current actual value Ch.10 <-> Data Pointer/CurrentActualValues[9]
//     Term 8 (AT2200-0500)/CC Inputs/Current actual value Ch.11 <-> Data Pointer/CurrentActualValues[10]
//     Term 8 (AT2200-0500)/CC Inputs/Current actual value Ch.12 <-> Data Pointer/CurrentActualValues[11]
//     Term 8 (AT2200-0500)/CC Inputs/Current actual value Ch.13 <-> Data Pointer/CurrentActualValues[12]
//     Term 8 (AT2200-0500)/CC Inputs/Current actual value Ch.14 <-> Data Pointer/CurrentActualValues[13]
//     Term 8 (AT2200-0500)/CC Inputs/Current actual value Ch.15 <-> Data Pointer/CurrentActualValues[14]
//     Term 8 (AT2200-0500)/CC Inputs/Current actual value Ch.16 <-> Data Pointer/CurrentActualValues[15]
//     Term 8 (AT2200-0500)/CC Inputs/Current actual value Ch.17 <-> Data Pointer/CurrentActualValues[16]
//     Term 8 (AT2200-0500)/CC Inputs/Current actual value Ch.18 <-> Data Pointer/CurrentActualValues[17]
//     Term 8 (AT2200-0500)/CC Inputs/Current actual value Ch.19 <-> Data Pointer/CurrentActualValues[18]
//     Term 8 (AT2200-0500)/CC Inputs/Current actual value Ch.2 <-> Data Pointer/CurrentActualValues[1]
//     Term 8 (AT2200-0500)/CC Inputs/Current actual value Ch.20 <-> Data Pointer/CurrentActualValues[19]
//     Term 8 (AT2200-0500)/CC Inputs/Current actual value Ch.21 <-> Data Pointer/CurrentActualValues[20]
//     Term 8 (AT2200-0500)/CC Inputs/Current actual value Ch.22 <-> Data Pointer/CurrentActualValues[21]
//     Term 8 (AT2200-0500)/CC Inputs/Current actual value Ch.23 <-> Data Pointer/CurrentActualValues[22]
//     Term 8 (AT2200-0500)/CC Inputs/Current actual value Ch.24 <-> Data Pointer/CurrentActualValues[23]
//     Term 8 (AT2200-0500)/CC Inputs/Current actual value Ch.25 <-> Data Pointer/CurrentActualValues[24]
//     Term 8 (AT2200-0500)/CC Inputs/Current actual value Ch.26 <-> Data Pointer/CurrentActualValues[25]
//     Term 8 (AT2200-0500)/CC Inputs/Current actual value Ch.27 <-> Data Pointer/CurrentActualValues[26]
//     Term 8 (AT2200-0500)/CC Inputs/Current actual value Ch.28 <-> Data Pointer/CurrentActualValues[27]
//     Term 8 (AT2200-0500)/CC Inputs/Current actual value Ch.29 <-> Data Pointer/CurrentActualValues[28]
//     Term 8 (AT2200-0500)/CC Inputs/Current actual value Ch.3 <-> Data Pointer/CurrentActualValues[2]
//     Term 8 (AT2200-0500)/CC Inputs/Current actual value Ch.30 <-> Data Pointer/CurrentActualValues[29]
//     Term 8 (AT2200-0500)/CC Inputs/Current actual value Ch.4 <-> Data Pointer/CurrentActualValues[3]
//     Term 8 (AT2200-0500)/CC Inputs/Current actual value Ch.5 <-> Data Pointer/CurrentActualValues[4]
//     Term 8 (AT2200-0500)/CC Inputs/Current actual value Ch.6 <-> Data Pointer/CurrentActualValues[5]
//     Term 8 (AT2200-0500)/CC Inputs/Current actual value Ch.7 <-> Data Pointer/CurrentActualValues[6]
//     Term 8 (AT2200-0500)/CC Inputs/Current actual value Ch.8 <-> Data Pointer/CurrentActualValues[7]
//     Term 8 (AT2200-0500)/CC Inputs/Current actual value Ch.9 <-> Data Pointer/CurrentActualValues[8]
//     Term 8 (AT2200-0500)/CC Inputs/Status <-> Data Pointer/Status
//     Term 8 (AT2200-0500)/CC Outputs/Control <-> Data Pointer/Control
//     Term 8 (AT2200-0500)/CC Outputs/Current setpoint value Ch.1 <-> Data Pointer/CurrentSetpointValues[0]
//     Term 8 (AT2200-0500)/CC Outputs/Current setpoint value Ch.10 <-> Data Pointer/CurrentSetpointValues[9]
//     Term 8 (AT2200-0500)/CC Outputs/Current setpoint value Ch.11 <-> Data Pointer/CurrentSetpointValues[10]
//     Term 8 (AT2200-0500)/CC Outputs/Current setpoint value Ch.12 <-> Data Pointer/CurrentSetpointValues[11]
//     Term 8 (AT2200-0500)/CC Outputs/Current setpoint value Ch.13 <-> Data Pointer/CurrentSetpointValues[12]
//     Term 8 (AT2200-0500)/CC Outputs/Current setpoint value Ch.14 <-> Data Pointer/CurrentSetpointValues[13]
//     Term 8 (AT2200-0500)/CC Outputs/Current setpoint value Ch.15 <-> Data Pointer/CurrentSetpointValues[14]
//     Term 8 (AT2200-0500)/CC Outputs/Current setpoint value Ch.16 <-> Data Pointer/CurrentSetpointValues[15]
//     Term 8 (AT2200-0500)/CC Outputs/Current setpoint value Ch.17 <-> Data Pointer/CurrentSetpointValues[16]
//     Term 8 (AT2200-0500)/CC Outputs/Current setpoint value Ch.18 <-> Data Pointer/CurrentSetpointValues[17]
//     Term 8 (AT2200-0500)/CC Outputs/Current setpoint value Ch.19 <-> Data Pointer/CurrentSetpointValues[18]
//     Term 8 (AT2200-0500)/CC Outputs/Current setpoint value Ch.2 <-> Data Pointer/CurrentSetpointValues[1]
//     Term 8 (AT2200-0500)/CC Outputs/Current setpoint value Ch.20 <-> Data Pointer/CurrentSetpointValues[19]
//     Term 8 (AT2200-0500)/CC Outputs/Current setpoint value Ch.21 <-> Data Pointer/CurrentSetpointValues[20]
//     Term 8 (AT2200-0500)/CC Outputs/Current setpoint value Ch.22 <-> Data Pointer/CurrentSetpointValues[21]
//     Term 8 (AT2200-0500)/CC Outputs/Current setpoint value Ch.23 <-> Data Pointer/CurrentSetpointValues[22]
//     Term 8 (AT2200-0500)/CC Outputs/Current setpoint value Ch.24 <-> Data Pointer/CurrentSetpointValues[23]
//     Term 8 (AT2200-0500)/CC Outputs/Current setpoint value Ch.25 <-> Data Pointer/CurrentSetpointValues[24]
//     Term 8 (AT2200-0500)/CC Outputs/Current setpoint value Ch.26 <-> Data Pointer/CurrentSetpointValues[25]
//     Term 8 (AT2200-0500)/CC Outputs/Current setpoint value Ch.27 <-> Data Pointer/CurrentSetpointValues[26]
//     Term 8 (AT2200-0500)/CC Outputs/Current setpoint value Ch.28 <-> Data Pointer/CurrentSetpointValues[27]
//     Term 8 (AT2200-0500)/CC Outputs/Current setpoint value Ch.29 <-> Data Pointer/CurrentSetpointValues[28]
//     Term 8 (AT2200-0500)/CC Outputs/Current setpoint value Ch.3 <-> Data Pointer/CurrentSetpointValues[2]
//     Term 8 (AT2200-0500)/CC Outputs/Current setpoint value Ch.30 <-> Data Pointer/CurrentSetpointValues[29]
//     Term 8 (AT2200-0500)/CC Outputs/Current setpoint value Ch.4 <-> Data Pointer/CurrentSetpointValues[3]
//     Term 8 (AT2200-0500)/CC Outputs/Current setpoint value Ch.5 <-> Data Pointer/CurrentSetpointValues[4]
//     Term 8 (AT2200-0500)/CC Outputs/Current setpoint value Ch.6 <-> Data Pointer/CurrentSetpointValues[5]
//     Term 8 (AT2200-0500)/CC Outputs/Current setpoint value Ch.7 <-> Data Pointer/CurrentSetpointValues[6]
//     Term 8 (AT2200-0500)/CC Outputs/Current setpoint value Ch.8 <-> Data Pointer/CurrentSetpointValues[7]
//     Term 8 (AT2200-0500)/CC Outputs/Current setpoint value Ch.9 <-> Data Pointer/CurrentSetpointValues[8]
//     Term 8 (AT2200-0500)/LFB Inputs/BinaryData <-> Data Pointer/HallSensorValues
//   Device 18 <-> TcCOM Objects/XTS ProcessingUnit 1/Part 1/Module 9
//     Term 9 (AT2040-0250)/CC Inputs/Current actual value Ch.1 <-> Data Pointer/CurrentActualValues[0]
//     Term 9 (AT2040-0250)/CC Inputs/Current actual value Ch.10 <-> Data Pointer/CurrentActualValues[9]
//     Term 9 (AT2040-0250)/CC Inputs/Current actual value Ch.11 <-> Data Pointer/CurrentActualValues[10]
//     Term 9 (AT2040-0250)/CC Inputs/Current actual value Ch.12 <-> Data Pointer/CurrentActualValues[11]
//     Term 9 (AT2040-0250)/CC Inputs/Current actual value Ch.13 <-> Data Pointer/CurrentActualValues[12]
//     Term 9 (AT2040-0250)/CC Inputs/Current actual value Ch.14 <-> Data Pointer/CurrentActualValues[13]
//     Term 9 (AT2040-0250)/CC Inputs/Current actual value Ch.15 <-> Data Pointer/CurrentActualValues[14]
//     Term 9 (AT2040-0250)/CC Inputs/Current actual value Ch.2 <-> Data Pointer/CurrentActualValues[1]
//     Term 9 (AT2040-0250)/CC Inputs/Current actual value Ch.3 <-> Data Pointer/CurrentActualValues[2]
//     Term 9 (AT2040-0250)/CC Inputs/Current actual value Ch.4 <-> Data Pointer/CurrentActualValues[3]
//     Term 9 (AT2040-0250)/CC Inputs/Current actual value Ch.5 <-> Data Pointer/CurrentActualValues[4]
//     Term 9 (AT2040-0250)/CC Inputs/Current actual value Ch.6 <-> Data Pointer/CurrentActualValues[5]
//     Term 9 (AT2040-0250)/CC Inputs/Current actual value Ch.7 <-> Data Pointer/CurrentActualValues[6]
//     Term 9 (AT2040-0250)/CC Inputs/Current actual value Ch.8 <-> Data Pointer/CurrentActualValues[7]
//     Term 9 (AT2040-0250)/CC Inputs/Current actual value Ch.9 <-> Data Pointer/CurrentActualValues[8]
//     Term 9 (AT2040-0250)/CC Inputs/Status <-> Data Pointer/Status
//     Term 9 (AT2040-0250)/CC Outputs/Control <-> Data Pointer/Control
//     Term 9 (AT2040-0250)/CC Outputs/Current setpoint value Ch.1 <-> Data Pointer/CurrentSetpointValues[0]
//     Term 9 (AT2040-0250)/CC Outputs/Current setpoint value Ch.10 <-> Data Pointer/CurrentSetpointValues[9]
//     Term 9 (AT2040-0250)/CC Outputs/Current setpoint value Ch.11 <-> Data Pointer/CurrentSetpointValues[10]
//     Term 9 (AT2040-0250)/CC Outputs/Current setpoint value Ch.12 <-> Data Pointer/CurrentSetpointValues[11]
//     Term 9 (AT2040-0250)/CC Outputs/Current setpoint value Ch.13 <-> Data Pointer/CurrentSetpointValues[12]
//     Term 9 (AT2040-0250)/CC Outputs/Current setpoint value Ch.14 <-> Data Pointer/CurrentSetpointValues[13]
//     Term 9 (AT2040-0250)/CC Outputs/Current setpoint value Ch.15 <-> Data Pointer/CurrentSetpointValues[14]
//     Term 9 (AT2040-0250)/CC Outputs/Current setpoint value Ch.2 <-> Data Pointer/CurrentSetpointValues[1]
//     Term 9 (AT2040-0250)/CC Outputs/Current setpoint value Ch.3 <-> Data Pointer/CurrentSetpointValues[2]
//     Term 9 (AT2040-0250)/CC Outputs/Current setpoint value Ch.4 <-> Data Pointer/CurrentSetpointValues[3]
//     Term 9 (AT2040-0250)/CC Outputs/Current setpoint value Ch.5 <-> Data Pointer/CurrentSetpointValues[4]
//     Term 9 (AT2040-0250)/CC Outputs/Current setpoint value Ch.6 <-> Data Pointer/CurrentSetpointValues[5]
//     Term 9 (AT2040-0250)/CC Outputs/Current setpoint value Ch.7 <-> Data Pointer/CurrentSetpointValues[6]
//     Term 9 (AT2040-0250)/CC Outputs/Current setpoint value Ch.8 <-> Data Pointer/CurrentSetpointValues[7]
//     Term 9 (AT2040-0250)/CC Outputs/Current setpoint value Ch.9 <-> Data Pointer/CurrentSetpointValues[8]
//     Term 9 (AT2040-0250)/Term 10 (AT2040-5250)/FB Inputs/Value Channel 01 <-> Data Pointer/RawPositionValues[0]
//     Term 9 (AT2040-0250)/Term 10 (AT2040-5250)/FB Inputs/Value Channel 02 <-> Data Pointer/RawPositionValues[1]
//     Term 9 (AT2040-0250)/Term 10 (AT2040-5250)/FB Inputs/Value Channel 03 <-> Data Pointer/RawPositionValues[2]
//     Term 9 (AT2040-0250)/Term 10 (AT2040-5250)/FB Inputs/Value Channel 04 <-> Data Pointer/RawPositionValues[3]
//     Term 9 (AT2040-0250)/Term 10 (AT2040-5250)/FB Inputs/Value Channel 05 <-> Data Pointer/RawPositionValues[4]
//     Term 9 (AT2040-0250)/Term 10 (AT2040-5250)/FB Inputs/Value Channel 06 <-> Data Pointer/RawPositionValues[5]
//     Term 9 (AT2040-0250)/Term 10 (AT2040-5250)/FB Inputs/Value Channel 07 <-> Data Pointer/RawPositionValues[6]
//     Term 9 (AT2040-0250)/Term 10 (AT2040-5250)/FB Inputs/Value Channel 08 <-> Data Pointer/RawPositionValues[7]
//     Term 9 (AT2040-0250)/Term 10 (AT2040-5250)/FB Inputs/Value Channel 09 <-> Data Pointer/RawPositionValues[8]
//     Term 9 (AT2040-0250)/Term 10 (AT2040-5250)/FB Inputs/Value Channel 10 <-> Data Pointer/RawPositionValues[9]
//     Term 9 (AT2040-0250)/Term 10 (AT2040-5250)/FB Inputs/Value Channel 11 <-> Data Pointer/RawPositionValues[10]
//     Term 9 (AT2040-0250)/Term 10 (AT2040-5250)/FB Inputs/Value Channel 12 <-> Data Pointer/RawPositionValues[11]
//     Term 9 (AT2040-0250)/Term 10 (AT2040-5250)/FB Inputs/Value Channel 13 <-> Data Pointer/RawPositionValues[12]
//     Term 9 (AT2040-0250)/Term 10 (AT2040-5250)/FB Inputs/Value Channel 14 <-> Data Pointer/RawPositionValues[13]
//     Term 9 (AT2040-0250)/Term 10 (AT2040-5250)/FB Inputs/Value Channel 15 <-> Data Pointer/RawPositionValues[14]
//     Term 9 (AT2040-0250)/Term 10 (AT2040-5250)/FB Inputs/Value Channel 16 <-> Data Pointer/RawPositionValues[15]
//     Term 9 (AT2040-0250)/Term 10 (AT2040-5250)/FB Inputs/Value Channel 17 <-> Data Pointer/RawPositionValues[16]
//     Term 9 (AT2040-0250)/Term 10 (AT2040-5250)/FB Inputs/Value Channel 18 <-> Data Pointer/RawPositionValues[17]
//     Term 9 (AT2040-0250)/Term 10 (AT2040-5250)/FB Inputs/Value Channel 19 <-> Data Pointer/RawPositionValues[18]
//     Term 9 (AT2040-0250)/Term 10 (AT2040-5250)/FB Inputs/Value Channel 20 <-> Data Pointer/RawPositionValues[19]
//     Term 9 (AT2040-0250)/Term 10 (AT2040-5250)/FB Inputs/Value Channel 21 <-> Data Pointer/RawPositionValues[20]
//     Term 9 (AT2040-0250)/Term 10 (AT2040-5250)/FB Inputs/Value Channel 22 <-> Data Pointer/RawPositionValues[21]
//     Term 9 (AT2040-0250)/Term 10 (AT2040-5250)/FB Inputs/Value Channel 23 <-> Data Pointer/RawPositionValues[22]
//     Term 9 (AT2040-0250)/Term 10 (AT2040-5250)/FB Inputs/Value Channel 24 <-> Data Pointer/RawPositionValues[23]
//     Term 9 (AT2040-0250)/Term 10 (AT2040-5250)/FB Inputs/Value Channel 25 <-> Data Pointer/RawPositionValues[24]
//     Term 9 (AT2040-0250)/Term 10 (AT2040-5250)/FB Inputs/Value Channel 26 <-> Data Pointer/RawPositionValues[25]
//     Term 9 (AT2040-0250)/Term 10 (AT2040-5250)/FB Inputs/Value Channel 27 <-> Data Pointer/RawPositionValues[26]
//     Term 9 (AT2040-0250)/Term 10 (AT2040-5250)/FB Inputs/Value Channel 28 <-> Data Pointer/RawPositionValues[27]
//     Term 9 (AT2040-0250)/Term 10 (AT2040-5250)/FB Inputs/Value Channel 29 <-> Data Pointer/RawPositionValues[28]
//     Term 9 (AT2040-0250)/Term 10 (AT2040-5250)/FB Inputs/Value Channel 30 <-> Data Pointer/RawPositionValues[29]
//     Term 9 (AT2040-0250)/Term 10 (AT2040-5250)/FB Inputs/Value Channel 31 <-> Data Pointer/RawPositionValues[30]
//     Term 9 (AT2040-0250)/Term 10 (AT2040-5250)/FB Inputs/Value Channel 32 <-> Data Pointer/RawPositionValues[31]
//   Device 19 <-> TcCOM Objects/XTS ProcessingUnit 1/Part 1/Module 11
//     Term 13 (AT2202-0500)/CC Inputs/Current actual value Ch.1 <-> Data Pointer/CurrentActualValues[0]
//     Term 13 (AT2202-0500)/CC Inputs/Current actual value Ch.10 <-> Data Pointer/CurrentActualValues[9]
//     Term 13 (AT2202-0500)/CC Inputs/Current actual value Ch.11 <-> Data Pointer/CurrentActualValues[10]
//     Term 13 (AT2202-0500)/CC Inputs/Current actual value Ch.12 <-> Data Pointer/CurrentActualValues[11]
//     Term 13 (AT2202-0500)/CC Inputs/Current actual value Ch.13 <-> Data Pointer/CurrentActualValues[12]
//     Term 13 (AT2202-0500)/CC Inputs/Current actual value Ch.14 <-> Data Pointer/CurrentActualValues[13]
//     Term 13 (AT2202-0500)/CC Inputs/Current actual value Ch.15 <-> Data Pointer/CurrentActualValues[14]
//     Term 13 (AT2202-0500)/CC Inputs/Current actual value Ch.16 <-> Data Pointer/CurrentActualValues[15]
//     Term 13 (AT2202-0500)/CC Inputs/Current actual value Ch.17 <-> Data Pointer/CurrentActualValues[16]
//     Term 13 (AT2202-0500)/CC Inputs/Current actual value Ch.18 <-> Data Pointer/CurrentActualValues[17]
//     Term 13 (AT2202-0500)/CC Inputs/Current actual value Ch.19 <-> Data Pointer/CurrentActualValues[18]
//     Term 13 (AT2202-0500)/CC Inputs/Current actual value Ch.2 <-> Data Pointer/CurrentActualValues[1]
//     Term 13 (AT2202-0500)/CC Inputs/Current actual value Ch.20 <-> Data Pointer/CurrentActualValues[19]
//     Term 13 (AT2202-0500)/CC Inputs/Current actual value Ch.21 <-> Data Pointer/CurrentActualValues[20]
//     Term 13 (AT2202-0500)/CC Inputs/Current actual value Ch.22 <-> Data Pointer/CurrentActualValues[21]
//     Term 13 (AT2202-0500)/CC Inputs/Current actual value Ch.23 <-> Data Pointer/CurrentActualValues[22]
//     Term 13 (AT2202-0500)/CC Inputs/Current actual value Ch.24 <-> Data Pointer/CurrentActualValues[23]
//     Term 13 (AT2202-0500)/CC Inputs/Current actual value Ch.25 <-> Data Pointer/CurrentActualValues[24]
//     Term 13 (AT2202-0500)/CC Inputs/Current actual value Ch.26 <-> Data Pointer/CurrentActualValues[25]
//     Term 13 (AT2202-0500)/CC Inputs/Current actual value Ch.27 <-> Data Pointer/CurrentActualValues[26]
//     Term 13 (AT2202-0500)/CC Inputs/Current actual value Ch.28 <-> Data Pointer/CurrentActualValues[27]
//     Term 13 (AT2202-0500)/CC Inputs/Current actual value Ch.29 <-> Data Pointer/CurrentActualValues[28]
//     Term 13 (AT2202-0500)/CC Inputs/Current actual value Ch.3 <-> Data Pointer/CurrentActualValues[2]
//     Term 13 (AT2202-0500)/CC Inputs/Current actual value Ch.30 <-> Data Pointer/CurrentActualValues[29]
//     Term 13 (AT2202-0500)/CC Inputs/Current actual value Ch.4 <-> Data Pointer/CurrentActualValues[3]
//     Term 13 (AT2202-0500)/CC Inputs/Current actual value Ch.5 <-> Data Pointer/CurrentActualValues[4]
//     Term 13 (AT2202-0500)/CC Inputs/Current actual value Ch.6 <-> Data Pointer/CurrentActualValues[5]
//     Term 13 (AT2202-0500)/CC Inputs/Current actual value Ch.7 <-> Data Pointer/CurrentActualValues[6]
//     Term 13 (AT2202-0500)/CC Inputs/Current actual value Ch.8 <-> Data Pointer/CurrentActualValues[7]
//     Term 13 (AT2202-0500)/CC Inputs/Current actual value Ch.9 <-> Data Pointer/CurrentActualValues[8]
//     Term 13 (AT2202-0500)/CC Inputs/Status <-> Data Pointer/Status
//     Term 13 (AT2202-0500)/CC Outputs/Control <-> Data Pointer/Control
//     Term 13 (AT2202-0500)/CC Outputs/Current setpoint value Ch.1 <-> Data Pointer/CurrentSetpointValues[0]
//     Term 13 (AT2202-0500)/CC Outputs/Current setpoint value Ch.10 <-> Data Pointer/CurrentSetpointValues[9]
//     Term 13 (AT2202-0500)/CC Outputs/Current setpoint value Ch.11 <-> Data Pointer/CurrentSetpointValues[10]
//     Term 13 (AT2202-0500)/CC Outputs/Current setpoint value Ch.12 <-> Data Pointer/CurrentSetpointValues[11]
//     Term 13 (AT2202-0500)/CC Outputs/Current setpoint value Ch.13 <-> Data Pointer/CurrentSetpointValues[12]
//     Term 13 (AT2202-0500)/CC Outputs/Current setpoint value Ch.14 <-> Data Pointer/CurrentSetpointValues[13]
//     Term 13 (AT2202-0500)/CC Outputs/Current setpoint value Ch.15 <-> Data Pointer/CurrentSetpointValues[14]
//     Term 13 (AT2202-0500)/CC Outputs/Current setpoint value Ch.16 <-> Data Pointer/CurrentSetpointValues[15]
//     Term 13 (AT2202-0500)/CC Outputs/Current setpoint value Ch.17 <-> Data Pointer/CurrentSetpointValues[16]
//     Term 13 (AT2202-0500)/CC Outputs/Current setpoint value Ch.18 <-> Data Pointer/CurrentSetpointValues[17]
//     Term 13 (AT2202-0500)/CC Outputs/Current setpoint value Ch.19 <-> Data Pointer/CurrentSetpointValues[18]
//     Term 13 (AT2202-0500)/CC Outputs/Current setpoint value Ch.2 <-> Data Pointer/CurrentSetpointValues[1]
//     Term 13 (AT2202-0500)/CC Outputs/Current setpoint value Ch.20 <-> Data Pointer/CurrentSetpointValues[19]
//     Term 13 (AT2202-0500)/CC Outputs/Current setpoint value Ch.21 <-> Data Pointer/CurrentSetpointValues[20]
//     Term 13 (AT2202-0500)/CC Outputs/Current setpoint value Ch.22 <-> Data Pointer/CurrentSetpointValues[21]
//     Term 13 (AT2202-0500)/CC Outputs/Current setpoint value Ch.23 <-> Data Pointer/CurrentSetpointValues[22]
//     Term 13 (AT2202-0500)/CC Outputs/Current setpoint value Ch.24 <-> Data Pointer/CurrentSetpointValues[23]
//     Term 13 (AT2202-0500)/CC Outputs/Current setpoint value Ch.25 <-> Data Pointer/CurrentSetpointValues[24]
//     Term 13 (AT2202-0500)/CC Outputs/Current setpoint value Ch.26 <-> Data Pointer/CurrentSetpointValues[25]
//     Term 13 (AT2202-0500)/CC Outputs/Current setpoint value Ch.27 <-> Data Pointer/CurrentSetpointValues[26]
//     Term 13 (AT2202-0500)/CC Outputs/Current setpoint value Ch.28 <-> Data Pointer/CurrentSetpointValues[27]
//     Term 13 (AT2202-0500)/CC Outputs/Current setpoint value Ch.29 <-> Data Pointer/CurrentSetpointValues[28]
//     Term 13 (AT2202-0500)/CC Outputs/Current setpoint value Ch.3 <-> Data Pointer/CurrentSetpointValues[2]
//     Term 13 (AT2202-0500)/CC Outputs/Current setpoint value Ch.30 <-> Data Pointer/CurrentSetpointValues[29]
//     Term 13 (AT2202-0500)/CC Outputs/Current setpoint value Ch.4 <-> Data Pointer/CurrentSetpointValues[3]
//     Term 13 (AT2202-0500)/CC Outputs/Current setpoint value Ch.5 <-> Data Pointer/CurrentSetpointValues[4]
//     Term 13 (AT2202-0500)/CC Outputs/Current setpoint value Ch.6 <-> Data Pointer/CurrentSetpointValues[5]
//     Term 13 (AT2202-0500)/CC Outputs/Current setpoint value Ch.7 <-> Data Pointer/CurrentSetpointValues[6]
//     Term 13 (AT2202-0500)/CC Outputs/Current setpoint value Ch.8 <-> Data Pointer/CurrentSetpointValues[7]
//     Term 13 (AT2202-0500)/CC Outputs/Current setpoint value Ch.9 <-> Data Pointer/CurrentSetpointValues[8]
//     Term 13 (AT2202-0500)/LFB Inputs/BinaryData <-> Data Pointer/HallSensorValues
//   Device 19 <-> TcCOM Objects/XTS ProcessingUnit 1/Part 1/Module 12
//     Term 14 (AT2200-0500)/CC Inputs/Current actual value Ch.1 <-> Data Pointer/CurrentActualValues[0]
//     Term 14 (AT2200-0500)/CC Inputs/Current actual value Ch.10 <-> Data Pointer/CurrentActualValues[9]
//     Term 14 (AT2200-0500)/CC Inputs/Current actual value Ch.11 <-> Data Pointer/CurrentActualValues[10]
//     Term 14 (AT2200-0500)/CC Inputs/Current actual value Ch.12 <-> Data Pointer/CurrentActualValues[11]
//     Term 14 (AT2200-0500)/CC Inputs/Current actual value Ch.13 <-> Data Pointer/CurrentActualValues[12]
//     Term 14 (AT2200-0500)/CC Inputs/Current actual value Ch.14 <-> Data Pointer/CurrentActualValues[13]
//     Term 14 (AT2200-0500)/CC Inputs/Current actual value Ch.15 <-> Data Pointer/CurrentActualValues[14]
//     Term 14 (AT2200-0500)/CC Inputs/Current actual value Ch.16 <-> Data Pointer/CurrentActualValues[15]
//     Term 14 (AT2200-0500)/CC Inputs/Current actual value Ch.17 <-> Data Pointer/CurrentActualValues[16]
//     Term 14 (AT2200-0500)/CC Inputs/Current actual value Ch.18 <-> Data Pointer/CurrentActualValues[17]
//     Term 14 (AT2200-0500)/CC Inputs/Current actual value Ch.19 <-> Data Pointer/CurrentActualValues[18]
//     Term 14 (AT2200-0500)/CC Inputs/Current actual value Ch.2 <-> Data Pointer/CurrentActualValues[1]
//     Term 14 (AT2200-0500)/CC Inputs/Current actual value Ch.20 <-> Data Pointer/CurrentActualValues[19]
//     Term 14 (AT2200-0500)/CC Inputs/Current actual value Ch.21 <-> Data Pointer/CurrentActualValues[20]
//     Term 14 (AT2200-0500)/CC Inputs/Current actual value Ch.22 <-> Data Pointer/CurrentActualValues[21]
//     Term 14 (AT2200-0500)/CC Inputs/Current actual value Ch.23 <-> Data Pointer/CurrentActualValues[22]
//     Term 14 (AT2200-0500)/CC Inputs/Current actual value Ch.24 <-> Data Pointer/CurrentActualValues[23]
//     Term 14 (AT2200-0500)/CC Inputs/Current actual value Ch.25 <-> Data Pointer/CurrentActualValues[24]
//     Term 14 (AT2200-0500)/CC Inputs/Current actual value Ch.26 <-> Data Pointer/CurrentActualValues[25]
//     Term 14 (AT2200-0500)/CC Inputs/Current actual value Ch.27 <-> Data Pointer/CurrentActualValues[26]
//     Term 14 (AT2200-0500)/CC Inputs/Current actual value Ch.28 <-> Data Pointer/CurrentActualValues[27]
//     Term 14 (AT2200-0500)/CC Inputs/Current actual value Ch.29 <-> Data Pointer/CurrentActualValues[28]
//     Term 14 (AT2200-0500)/CC Inputs/Current actual value Ch.3 <-> Data Pointer/CurrentActualValues[2]
//     Term 14 (AT2200-0500)/CC Inputs/Current actual value Ch.30 <-> Data Pointer/CurrentActualValues[29]
//     Term 14 (AT2200-0500)/CC Inputs/Current actual value Ch.4 <-> Data Pointer/CurrentActualValues[3]
//     Term 14 (AT2200-0500)/CC Inputs/Current actual value Ch.5 <-> Data Pointer/CurrentActualValues[4]
//     Term 14 (AT2200-0500)/CC Inputs/Current actual value Ch.6 <-> Data Pointer/CurrentActualValues[5]
//     Term 14 (AT2200-0500)/CC Inputs/Current actual value Ch.7 <-> Data Pointer/CurrentActualValues[6]
//     Term 14 (AT2200-0500)/CC Inputs/Current actual value Ch.8 <-> Data Pointer/CurrentActualValues[7]
//     Term 14 (AT2200-0500)/CC Inputs/Current actual value Ch.9 <-> Data Pointer/CurrentActualValues[8]
//     Term 14 (AT2200-0500)/CC Inputs/Status <-> Data Pointer/Status
//     Term 14 (AT2200-0500)/CC Outputs/Control <-> Data Pointer/Control
//     Term 14 (AT2200-0500)/CC Outputs/Current setpoint value Ch.1 <-> Data Pointer/CurrentSetpointValues[0]
//     Term 14 (AT2200-0500)/CC Outputs/Current setpoint value Ch.10 <-> Data Pointer/CurrentSetpointValues[9]
//     Term 14 (AT2200-0500)/CC Outputs/Current setpoint value Ch.11 <-> Data Pointer/CurrentSetpointValues[10]
//     Term 14 (AT2200-0500)/CC Outputs/Current setpoint value Ch.12 <-> Data Pointer/CurrentSetpointValues[11]
//     Term 14 (AT2200-0500)/CC Outputs/Current setpoint value Ch.13 <-> Data Pointer/CurrentSetpointValues[12]
//     Term 14 (AT2200-0500)/CC Outputs/Current setpoint value Ch.14 <-> Data Pointer/CurrentSetpointValues[13]
//     Term 14 (AT2200-0500)/CC Outputs/Current setpoint value Ch.15 <-> Data Pointer/CurrentSetpointValues[14]
//     Term 14 (AT2200-0500)/CC Outputs/Current setpoint value Ch.16 <-> Data Pointer/CurrentSetpointValues[15]
//     Term 14 (AT2200-0500)/CC Outputs/Current setpoint value Ch.17 <-> Data Pointer/CurrentSetpointValues[16]
//     Term 14 (AT2200-0500)/CC Outputs/Current setpoint value Ch.18 <-> Data Pointer/CurrentSetpointValues[17]
//     Term 14 (AT2200-0500)/CC Outputs/Current setpoint value Ch.19 <-> Data Pointer/CurrentSetpointValues[18]
//     Term 14 (AT2200-0500)/CC Outputs/Current setpoint value Ch.2 <-> Data Pointer/CurrentSetpointValues[1]
//     Term 14 (AT2200-0500)/CC Outputs/Current setpoint value Ch.20 <-> Data Pointer/CurrentSetpointValues[19]
//     Term 14 (AT2200-0500)/CC Outputs/Current setpoint value Ch.21 <-> Data Pointer/CurrentSetpointValues[20]
//     Term 14 (AT2200-0500)/CC Outputs/Current setpoint value Ch.22 <-> Data Pointer/CurrentSetpointValues[21]
//     Term 14 (AT2200-0500)/CC Outputs/Current setpoint value Ch.23 <-> Data Pointer/CurrentSetpointValues[22]
//     Term 14 (AT2200-0500)/CC Outputs/Current setpoint value Ch.24 <-> Data Pointer/CurrentSetpointValues[23]
//     Term 14 (AT2200-0500)/CC Outputs/Current setpoint value Ch.25 <-> Data Pointer/CurrentSetpointValues[24]
//     Term 14 (AT2200-0500)/CC Outputs/Current setpoint value Ch.26 <-> Data Pointer/CurrentSetpointValues[25]
//     Term 14 (AT2200-0500)/CC Outputs/Current setpoint value Ch.27 <-> Data Pointer/CurrentSetpointValues[26]
//     Term 14 (AT2200-0500)/CC Outputs/Current setpoint value Ch.28 <-> Data Pointer/CurrentSetpointValues[27]
//     Term 14 (AT2200-0500)/CC Outputs/Current setpoint value Ch.29 <-> Data Pointer/CurrentSetpointValues[28]
//     Term 14 (AT2200-0500)/CC Outputs/Current setpoint value Ch.3 <-> Data Pointer/CurrentSetpointValues[2]
//     Term 14 (AT2200-0500)/CC Outputs/Current setpoint value Ch.30 <-> Data Pointer/CurrentSetpointValues[29]
//     Term 14 (AT2200-0500)/CC Outputs/Current setpoint value Ch.4 <-> Data Pointer/CurrentSetpointValues[3]
//     Term 14 (AT2200-0500)/CC Outputs/Current setpoint value Ch.5 <-> Data Pointer/CurrentSetpointValues[4]
//     Term 14 (AT2200-0500)/CC Outputs/Current setpoint value Ch.6 <-> Data Pointer/CurrentSetpointValues[5]
//     Term 14 (AT2200-0500)/CC Outputs/Current setpoint value Ch.7 <-> Data Pointer/CurrentSetpointValues[6]
//     Term 14 (AT2200-0500)/CC Outputs/Current setpoint value Ch.8 <-> Data Pointer/CurrentSetpointValues[7]
//     Term 14 (AT2200-0500)/CC Outputs/Current setpoint value Ch.9 <-> Data Pointer/CurrentSetpointValues[8]
//     Term 14 (AT2200-0500)/LFB Inputs/BinaryData <-> Data Pointer/HallSensorValues
//   Device 19 <-> TcCOM Objects/XTS ProcessingUnit 1/Part 1/Module 13
//     Term 15 (AT2000-0250)/CC Inputs/Current actual value Ch.1 <-> Data Pointer/CurrentActualValues[0]
//     Term 15 (AT2000-0250)/CC Inputs/Current actual value Ch.10 <-> Data Pointer/CurrentActualValues[9]
//     Term 15 (AT2000-0250)/CC Inputs/Current actual value Ch.11 <-> Data Pointer/CurrentActualValues[10]
//     Term 15 (AT2000-0250)/CC Inputs/Current actual value Ch.12 <-> Data Pointer/CurrentActualValues[11]
//     Term 15 (AT2000-0250)/CC Inputs/Current actual value Ch.13 <-> Data Pointer/CurrentActualValues[12]
//     Term 15 (AT2000-0250)/CC Inputs/Current actual value Ch.14 <-> Data Pointer/CurrentActualValues[13]
//     Term 15 (AT2000-0250)/CC Inputs/Current actual value Ch.15 <-> Data Pointer/CurrentActualValues[14]
//     Term 15 (AT2000-0250)/CC Inputs/Current actual value Ch.2 <-> Data Pointer/CurrentActualValues[1]
//     Term 15 (AT2000-0250)/CC Inputs/Current actual value Ch.3 <-> Data Pointer/CurrentActualValues[2]
//     Term 15 (AT2000-0250)/CC Inputs/Current actual value Ch.4 <-> Data Pointer/CurrentActualValues[3]
//     Term 15 (AT2000-0250)/CC Inputs/Current actual value Ch.5 <-> Data Pointer/CurrentActualValues[4]
//     Term 15 (AT2000-0250)/CC Inputs/Current actual value Ch.6 <-> Data Pointer/CurrentActualValues[5]
//     Term 15 (AT2000-0250)/CC Inputs/Current actual value Ch.7 <-> Data Pointer/CurrentActualValues[6]
//     Term 15 (AT2000-0250)/CC Inputs/Current actual value Ch.8 <-> Data Pointer/CurrentActualValues[7]
//     Term 15 (AT2000-0250)/CC Inputs/Current actual value Ch.9 <-> Data Pointer/CurrentActualValues[8]
//     Term 15 (AT2000-0250)/CC Inputs/Status <-> Data Pointer/Status
//     Term 15 (AT2000-0250)/CC Outputs/Control <-> Data Pointer/Control
//     Term 15 (AT2000-0250)/CC Outputs/Current setpoint value Ch.1 <-> Data Pointer/CurrentSetpointValues[0]
//     Term 15 (AT2000-0250)/CC Outputs/Current setpoint value Ch.10 <-> Data Pointer/CurrentSetpointValues[9]
//     Term 15 (AT2000-0250)/CC Outputs/Current setpoint value Ch.11 <-> Data Pointer/CurrentSetpointValues[10]
//     Term 15 (AT2000-0250)/CC Outputs/Current setpoint value Ch.12 <-> Data Pointer/CurrentSetpointValues[11]
//     Term 15 (AT2000-0250)/CC Outputs/Current setpoint value Ch.13 <-> Data Pointer/CurrentSetpointValues[12]
//     Term 15 (AT2000-0250)/CC Outputs/Current setpoint value Ch.14 <-> Data Pointer/CurrentSetpointValues[13]
//     Term 15 (AT2000-0250)/CC Outputs/Current setpoint value Ch.15 <-> Data Pointer/CurrentSetpointValues[14]
//     Term 15 (AT2000-0250)/CC Outputs/Current setpoint value Ch.2 <-> Data Pointer/CurrentSetpointValues[1]
//     Term 15 (AT2000-0250)/CC Outputs/Current setpoint value Ch.3 <-> Data Pointer/CurrentSetpointValues[2]
//     Term 15 (AT2000-0250)/CC Outputs/Current setpoint value Ch.4 <-> Data Pointer/CurrentSetpointValues[3]
//     Term 15 (AT2000-0250)/CC Outputs/Current setpoint value Ch.5 <-> Data Pointer/CurrentSetpointValues[4]
//     Term 15 (AT2000-0250)/CC Outputs/Current setpoint value Ch.6 <-> Data Pointer/CurrentSetpointValues[5]
//     Term 15 (AT2000-0250)/CC Outputs/Current setpoint value Ch.7 <-> Data Pointer/CurrentSetpointValues[6]
//     Term 15 (AT2000-0250)/CC Outputs/Current setpoint value Ch.8 <-> Data Pointer/CurrentSetpointValues[7]
//     Term 15 (AT2000-0250)/CC Outputs/Current setpoint value Ch.9 <-> Data Pointer/CurrentSetpointValues[8]
//     Term 15 (AT2000-0250)/Term 16 (AT2000-5250)/FB Inputs/Value Channel 01 <-> Data Pointer/RawPositionValues[0]
//     Term 15 (AT2000-0250)/Term 16 (AT2000-5250)/FB Inputs/Value Channel 02 <-> Data Pointer/RawPositionValues[1]
//     Term 15 (AT2000-0250)/Term 16 (AT2000-5250)/FB Inputs/Value Channel 03 <-> Data Pointer/RawPositionValues[2]
//     Term 15 (AT2000-0250)/Term 16 (AT2000-5250)/FB Inputs/Value Channel 04 <-> Data Pointer/RawPositionValues[3]
//     Term 15 (AT2000-0250)/Term 16 (AT2000-5250)/FB Inputs/Value Channel 05 <-> Data Pointer/RawPositionValues[4]
//     Term 15 (AT2000-0250)/Term 16 (AT2000-5250)/FB Inputs/Value Channel 06 <-> Data Pointer/RawPositionValues[5]
//     Term 15 (AT2000-0250)/Term 16 (AT2000-5250)/FB Inputs/Value Channel 07 <-> Data Pointer/RawPositionValues[6]
//     Term 15 (AT2000-0250)/Term 16 (AT2000-5250)/FB Inputs/Value Channel 08 <-> Data Pointer/RawPositionValues[7]
//     Term 15 (AT2000-0250)/Term 16 (AT2000-5250)/FB Inputs/Value Channel 09 <-> Data Pointer/RawPositionValues[8]
//     Term 15 (AT2000-0250)/Term 16 (AT2000-5250)/FB Inputs/Value Channel 10 <-> Data Pointer/RawPositionValues[9]
//     Term 15 (AT2000-0250)/Term 16 (AT2000-5250)/FB Inputs/Value Channel 11 <-> Data Pointer/RawPositionValues[10]
//     Term 15 (AT2000-0250)/Term 16 (AT2000-5250)/FB Inputs/Value Channel 12 <-> Data Pointer/RawPositionValues[11]
//     Term 15 (AT2000-0250)/Term 16 (AT2000-5250)/FB Inputs/Value Channel 13 <-> Data Pointer/RawPositionValues[12]
//     Term 15 (AT2000-0250)/Term 16 (AT2000-5250)/FB Inputs/Value Channel 14 <-> Data Pointer/RawPositionValues[13]
//     Term 15 (AT2000-0250)/Term 16 (AT2000-5250)/FB Inputs/Value Channel 15 <-> Data Pointer/RawPositionValues[14]
//     Term 15 (AT2000-0250)/Term 16 (AT2000-5250)/FB Inputs/Value Channel 16 <-> Data Pointer/RawPositionValues[15]
//     Term 15 (AT2000-0250)/Term 16 (AT2000-5250)/FB Inputs/Value Channel 17 <-> Data Pointer/RawPositionValues[16]
//     Term 15 (AT2000-0250)/Term 16 (AT2000-5250)/FB Inputs/Value Channel 18 <-> Data Pointer/RawPositionValues[17]
//     Term 15 (AT2000-0250)/Term 16 (AT2000-5250)/FB Inputs/Value Channel 19 <-> Data Pointer/RawPositionValues[18]
//     Term 15 (AT2000-0250)/Term 16 (AT2000-5250)/FB Inputs/Value Channel 20 <-> Data Pointer/RawPositionValues[19]
//     Term 15 (AT2000-0250)/Term 16 (AT2000-5250)/FB Inputs/Value Channel 21 <-> Data Pointer/RawPositionValues[20]
//     Term 15 (AT2000-0250)/Term 16 (AT2000-5250)/FB Inputs/Value Channel 22 <-> Data Pointer/RawPositionValues[21]
//     Term 15 (AT2000-0250)/Term 16 (AT2000-5250)/FB Inputs/Value Channel 23 <-> Data Pointer/RawPositionValues[22]
//     Term 15 (AT2000-0250)/Term 16 (AT2000-5250)/FB Inputs/Value Channel 24 <-> Data Pointer/RawPositionValues[23]
//     Term 15 (AT2000-0250)/Term 16 (AT2000-5250)/FB Inputs/Value Channel 25 <-> Data Pointer/RawPositionValues[24]
//     Term 15 (AT2000-0250)/Term 16 (AT2000-5250)/FB Inputs/Value Channel 26 <-> Data Pointer/RawPositionValues[25]
//     Term 15 (AT2000-0250)/Term 16 (AT2000-5250)/FB Inputs/Value Channel 27 <-> Data Pointer/RawPositionValues[26]
//     Term 15 (AT2000-0250)/Term 16 (AT2000-5250)/FB Inputs/Value Channel 28 <-> Data Pointer/RawPositionValues[27]
//     Term 15 (AT2000-0250)/Term 16 (AT2000-5250)/FB Inputs/Value Channel 29 <-> Data Pointer/RawPositionValues[28]
//     Term 15 (AT2000-0250)/Term 16 (AT2000-5250)/FB Inputs/Value Channel 30 <-> Data Pointer/RawPositionValues[29]
//     Term 15 (AT2000-0250)/Term 16 (AT2000-5250)/FB Inputs/Value Channel 31 <-> Data Pointer/RawPositionValues[30]
//     Term 15 (AT2000-0250)/Term 16 (AT2000-5250)/FB Inputs/Value Channel 32 <-> Data Pointer/RawPositionValues[31]
//   Device 20 <-> TcCOM Objects/XTS ProcessingUnit 1/Part 1/Module 14
//     Term 17 (AT2002-0250)/CC Inputs/Current actual value Ch.1 <-> Data Pointer/CurrentActualValues[0]
//     Term 17 (AT2002-0250)/CC Inputs/Current actual value Ch.10 <-> Data Pointer/CurrentActualValues[9]
//     Term 17 (AT2002-0250)/CC Inputs/Current actual value Ch.11 <-> Data Pointer/CurrentActualValues[10]
//     Term 17 (AT2002-0250)/CC Inputs/Current actual value Ch.12 <-> Data Pointer/CurrentActualValues[11]
//     Term 17 (AT2002-0250)/CC Inputs/Current actual value Ch.13 <-> Data Pointer/CurrentActualValues[12]
//     Term 17 (AT2002-0250)/CC Inputs/Current actual value Ch.14 <-> Data Pointer/CurrentActualValues[13]
//     Term 17 (AT2002-0250)/CC Inputs/Current actual value Ch.15 <-> Data Pointer/CurrentActualValues[14]
//     Term 17 (AT2002-0250)/CC Inputs/Current actual value Ch.2 <-> Data Pointer/CurrentActualValues[1]
//     Term 17 (AT2002-0250)/CC Inputs/Current actual value Ch.3 <-> Data Pointer/CurrentActualValues[2]
//     Term 17 (AT2002-0250)/CC Inputs/Current actual value Ch.4 <-> Data Pointer/CurrentActualValues[3]
//     Term 17 (AT2002-0250)/CC Inputs/Current actual value Ch.5 <-> Data Pointer/CurrentActualValues[4]
//     Term 17 (AT2002-0250)/CC Inputs/Current actual value Ch.6 <-> Data Pointer/CurrentActualValues[5]
//     Term 17 (AT2002-0250)/CC Inputs/Current actual value Ch.7 <-> Data Pointer/CurrentActualValues[6]
//     Term 17 (AT2002-0250)/CC Inputs/Current actual value Ch.8 <-> Data Pointer/CurrentActualValues[7]
//     Term 17 (AT2002-0250)/CC Inputs/Current actual value Ch.9 <-> Data Pointer/CurrentActualValues[8]
//     Term 17 (AT2002-0250)/CC Inputs/Status <-> Data Pointer/Status
//     Term 17 (AT2002-0250)/CC Outputs/Control <-> Data Pointer/Control
//     Term 17 (AT2002-0250)/CC Outputs/Current setpoint value Ch.1 <-> Data Pointer/CurrentSetpointValues[0]
//     Term 17 (AT2002-0250)/CC Outputs/Current setpoint value Ch.10 <-> Data Pointer/CurrentSetpointValues[9]
//     Term 17 (AT2002-0250)/CC Outputs/Current setpoint value Ch.11 <-> Data Pointer/CurrentSetpointValues[10]
//     Term 17 (AT2002-0250)/CC Outputs/Current setpoint value Ch.12 <-> Data Pointer/CurrentSetpointValues[11]
//     Term 17 (AT2002-0250)/CC Outputs/Current setpoint value Ch.13 <-> Data Pointer/CurrentSetpointValues[12]
//     Term 17 (AT2002-0250)/CC Outputs/Current setpoint value Ch.14 <-> Data Pointer/CurrentSetpointValues[13]
//     Term 17 (AT2002-0250)/CC Outputs/Current setpoint value Ch.15 <-> Data Pointer/CurrentSetpointValues[14]
//     Term 17 (AT2002-0250)/CC Outputs/Current setpoint value Ch.2 <-> Data Pointer/CurrentSetpointValues[1]
//     Term 17 (AT2002-0250)/CC Outputs/Current setpoint value Ch.3 <-> Data Pointer/CurrentSetpointValues[2]
//     Term 17 (AT2002-0250)/CC Outputs/Current setpoint value Ch.4 <-> Data Pointer/CurrentSetpointValues[3]
//     Term 17 (AT2002-0250)/CC Outputs/Current setpoint value Ch.5 <-> Data Pointer/CurrentSetpointValues[4]
//     Term 17 (AT2002-0250)/CC Outputs/Current setpoint value Ch.6 <-> Data Pointer/CurrentSetpointValues[5]
//     Term 17 (AT2002-0250)/CC Outputs/Current setpoint value Ch.7 <-> Data Pointer/CurrentSetpointValues[6]
//     Term 17 (AT2002-0250)/CC Outputs/Current setpoint value Ch.8 <-> Data Pointer/CurrentSetpointValues[7]
//     Term 17 (AT2002-0250)/CC Outputs/Current setpoint value Ch.9 <-> Data Pointer/CurrentSetpointValues[8]
//     Term 17 (AT2002-0250)/Term 18 (AT2002-5250)/FB Inputs/Value Channel 01 <-> Data Pointer/RawPositionValues[0]
//     Term 17 (AT2002-0250)/Term 18 (AT2002-5250)/FB Inputs/Value Channel 02 <-> Data Pointer/RawPositionValues[1]
//     Term 17 (AT2002-0250)/Term 18 (AT2002-5250)/FB Inputs/Value Channel 03 <-> Data Pointer/RawPositionValues[2]
//     Term 17 (AT2002-0250)/Term 18 (AT2002-5250)/FB Inputs/Value Channel 04 <-> Data Pointer/RawPositionValues[3]
//     Term 17 (AT2002-0250)/Term 18 (AT2002-5250)/FB Inputs/Value Channel 05 <-> Data Pointer/RawPositionValues[4]
//     Term 17 (AT2002-0250)/Term 18 (AT2002-5250)/FB Inputs/Value Channel 06 <-> Data Pointer/RawPositionValues[5]
//     Term 17 (AT2002-0250)/Term 18 (AT2002-5250)/FB Inputs/Value Channel 07 <-> Data Pointer/RawPositionValues[6]
//     Term 17 (AT2002-0250)/Term 18 (AT2002-5250)/FB Inputs/Value Channel 08 <-> Data Pointer/RawPositionValues[7]
//     Term 17 (AT2002-0250)/Term 18 (AT2002-5250)/FB Inputs/Value Channel 09 <-> Data Pointer/RawPositionValues[8]
//     Term 17 (AT2002-0250)/Term 18 (AT2002-5250)/FB Inputs/Value Channel 10 <-> Data Pointer/RawPositionValues[9]
//     Term 17 (AT2002-0250)/Term 18 (AT2002-5250)/FB Inputs/Value Channel 11 <-> Data Pointer/RawPositionValues[10]
//     Term 17 (AT2002-0250)/Term 18 (AT2002-5250)/FB Inputs/Value Channel 12 <-> Data Pointer/RawPositionValues[11]
//     Term 17 (AT2002-0250)/Term 18 (AT2002-5250)/FB Inputs/Value Channel 13 <-> Data Pointer/RawPositionValues[12]
//     Term 17 (AT2002-0250)/Term 18 (AT2002-5250)/FB Inputs/Value Channel 14 <-> Data Pointer/RawPositionValues[13]
//     Term 17 (AT2002-0250)/Term 18 (AT2002-5250)/FB Inputs/Value Channel 15 <-> Data Pointer/RawPositionValues[14]
//     Term 17 (AT2002-0250)/Term 18 (AT2002-5250)/FB Inputs/Value Channel 16 <-> Data Pointer/RawPositionValues[15]
//     Term 17 (AT2002-0250)/Term 18 (AT2002-5250)/FB Inputs/Value Channel 17 <-> Data Pointer/RawPositionValues[16]
//     Term 17 (AT2002-0250)/Term 18 (AT2002-5250)/FB Inputs/Value Channel 18 <-> Data Pointer/RawPositionValues[17]
//     Term 17 (AT2002-0250)/Term 18 (AT2002-5250)/FB Inputs/Value Channel 19 <-> Data Pointer/RawPositionValues[18]
//     Term 17 (AT2002-0250)/Term 18 (AT2002-5250)/FB Inputs/Value Channel 20 <-> Data Pointer/RawPositionValues[19]
//     Term 17 (AT2002-0250)/Term 18 (AT2002-5250)/FB Inputs/Value Channel 21 <-> Data Pointer/RawPositionValues[20]
//     Term 17 (AT2002-0250)/Term 18 (AT2002-5250)/FB Inputs/Value Channel 22 <-> Data Pointer/RawPositionValues[21]
//     Term 17 (AT2002-0250)/Term 18 (AT2002-5250)/FB Inputs/Value Channel 23 <-> Data Pointer/RawPositionValues[22]
//     Term 17 (AT2002-0250)/Term 18 (AT2002-5250)/FB Inputs/Value Channel 24 <-> Data Pointer/RawPositionValues[23]
//     Term 17 (AT2002-0250)/Term 18 (AT2002-5250)/FB Inputs/Value Channel 25 <-> Data Pointer/RawPositionValues[24]
//     Term 17 (AT2002-0250)/Term 18 (AT2002-5250)/FB Inputs/Value Channel 26 <-> Data Pointer/RawPositionValues[25]
//     Term 17 (AT2002-0250)/Term 18 (AT2002-5250)/FB Inputs/Value Channel 27 <-> Data Pointer/RawPositionValues[26]
//     Term 17 (AT2002-0250)/Term 18 (AT2002-5250)/FB Inputs/Value Channel 28 <-> Data Pointer/RawPositionValues[27]
//     Term 17 (AT2002-0250)/Term 18 (AT2002-5250)/FB Inputs/Value Channel 29 <-> Data Pointer/RawPositionValues[28]
//     Term 17 (AT2002-0250)/Term 18 (AT2002-5250)/FB Inputs/Value Channel 30 <-> Data Pointer/RawPositionValues[29]
//     Term 17 (AT2002-0250)/Term 18 (AT2002-5250)/FB Inputs/Value Channel 31 <-> Data Pointer/RawPositionValues[30]
//     Term 17 (AT2002-0250)/Term 18 (AT2002-5250)/FB Inputs/Value Channel 32 <-> Data Pointer/RawPositionValues[31]
//   Device 20 <-> TcCOM Objects/XTS ProcessingUnit 1/Part 1/Module 15
//     Term 19 (AT2200-0500)/CC Inputs/Current actual value Ch.1 <-> Data Pointer/CurrentActualValues[0]
//     Term 19 (AT2200-0500)/CC Inputs/Current actual value Ch.10 <-> Data Pointer/CurrentActualValues[9]
//     Term 19 (AT2200-0500)/CC Inputs/Current actual value Ch.11 <-> Data Pointer/CurrentActualValues[10]
//     Term 19 (AT2200-0500)/CC Inputs/Current actual value Ch.12 <-> Data Pointer/CurrentActualValues[11]
//     Term 19 (AT2200-0500)/CC Inputs/Current actual value Ch.13 <-> Data Pointer/CurrentActualValues[12]
//     Term 19 (AT2200-0500)/CC Inputs/Current actual value Ch.14 <-> Data Pointer/CurrentActualValues[13]
//     Term 19 (AT2200-0500)/CC Inputs/Current actual value Ch.15 <-> Data Pointer/CurrentActualValues[14]
//     Term 19 (AT2200-0500)/CC Inputs/Current actual value Ch.16 <-> Data Pointer/CurrentActualValues[15]
//     Term 19 (AT2200-0500)/CC Inputs/Current actual value Ch.17 <-> Data Pointer/CurrentActualValues[16]
//     Term 19 (AT2200-0500)/CC Inputs/Current actual value Ch.18 <-> Data Pointer/CurrentActualValues[17]
//     Term 19 (AT2200-0500)/CC Inputs/Current actual value Ch.19 <-> Data Pointer/CurrentActualValues[18]
//     Term 19 (AT2200-0500)/CC Inputs/Current actual value Ch.2 <-> Data Pointer/CurrentActualValues[1]
//     Term 19 (AT2200-0500)/CC Inputs/Current actual value Ch.20 <-> Data Pointer/CurrentActualValues[19]
//     Term 19 (AT2200-0500)/CC Inputs/Current actual value Ch.21 <-> Data Pointer/CurrentActualValues[20]
//     Term 19 (AT2200-0500)/CC Inputs/Current actual value Ch.22 <-> Data Pointer/CurrentActualValues[21]
//     Term 19 (AT2200-0500)/CC Inputs/Current actual value Ch.23 <-> Data Pointer/CurrentActualValues[22]
//     Term 19 (AT2200-0500)/CC Inputs/Current actual value Ch.24 <-> Data Pointer/CurrentActualValues[23]
//     Term 19 (AT2200-0500)/CC Inputs/Current actual value Ch.25 <-> Data Pointer/CurrentActualValues[24]
//     Term 19 (AT2200-0500)/CC Inputs/Current actual value Ch.26 <-> Data Pointer/CurrentActualValues[25]
//     Term 19 (AT2200-0500)/CC Inputs/Current actual value Ch.27 <-> Data Pointer/CurrentActualValues[26]
//     Term 19 (AT2200-0500)/CC Inputs/Current actual value Ch.28 <-> Data Pointer/CurrentActualValues[27]
//     Term 19 (AT2200-0500)/CC Inputs/Current actual value Ch.29 <-> Data Pointer/CurrentActualValues[28]
//     Term 19 (AT2200-0500)/CC Inputs/Current actual value Ch.3 <-> Data Pointer/CurrentActualValues[2]
//     Term 19 (AT2200-0500)/CC Inputs/Current actual value Ch.30 <-> Data Pointer/CurrentActualValues[29]
//     Term 19 (AT2200-0500)/CC Inputs/Current actual value Ch.4 <-> Data Pointer/CurrentActualValues[3]
//     Term 19 (AT2200-0500)/CC Inputs/Current actual value Ch.5 <-> Data Pointer/CurrentActualValues[4]
//     Term 19 (AT2200-0500)/CC Inputs/Current actual value Ch.6 <-> Data Pointer/CurrentActualValues[5]
//     Term 19 (AT2200-0500)/CC Inputs/Current actual value Ch.7 <-> Data Pointer/CurrentActualValues[6]
//     Term 19 (AT2200-0500)/CC Inputs/Current actual value Ch.8 <-> Data Pointer/CurrentActualValues[7]
//     Term 19 (AT2200-0500)/CC Inputs/Current actual value Ch.9 <-> Data Pointer/CurrentActualValues[8]
//     Term 19 (AT2200-0500)/CC Inputs/Status <-> Data Pointer/Status
//     Term 19 (AT2200-0500)/CC Outputs/Control <-> Data Pointer/Control
//     Term 19 (AT2200-0500)/CC Outputs/Current setpoint value Ch.1 <-> Data Pointer/CurrentSetpointValues[0]
//     Term 19 (AT2200-0500)/CC Outputs/Current setpoint value Ch.10 <-> Data Pointer/CurrentSetpointValues[9]
//     Term 19 (AT2200-0500)/CC Outputs/Current setpoint value Ch.11 <-> Data Pointer/CurrentSetpointValues[10]
//     Term 19 (AT2200-0500)/CC Outputs/Current setpoint value Ch.12 <-> Data Pointer/CurrentSetpointValues[11]
//     Term 19 (AT2200-0500)/CC Outputs/Current setpoint value Ch.13 <-> Data Pointer/CurrentSetpointValues[12]
//     Term 19 (AT2200-0500)/CC Outputs/Current setpoint value Ch.14 <-> Data Pointer/CurrentSetpointValues[13]
//     Term 19 (AT2200-0500)/CC Outputs/Current setpoint value Ch.15 <-> Data Pointer/CurrentSetpointValues[14]
//     Term 19 (AT2200-0500)/CC Outputs/Current setpoint value Ch.16 <-> Data Pointer/CurrentSetpointValues[15]
//     Term 19 (AT2200-0500)/CC Outputs/Current setpoint value Ch.17 <-> Data Pointer/CurrentSetpointValues[16]
//     Term 19 (AT2200-0500)/CC Outputs/Current setpoint value Ch.18 <-> Data Pointer/CurrentSetpointValues[17]
//     Term 19 (AT2200-0500)/CC Outputs/Current setpoint value Ch.19 <-> Data Pointer/CurrentSetpointValues[18]
//     Term 19 (AT2200-0500)/CC Outputs/Current setpoint value Ch.2 <-> Data Pointer/CurrentSetpointValues[1]
//     Term 19 (AT2200-0500)/CC Outputs/Current setpoint value Ch.20 <-> Data Pointer/CurrentSetpointValues[19]
//     Term 19 (AT2200-0500)/CC Outputs/Current setpoint value Ch.21 <-> Data Pointer/CurrentSetpointValues[20]
//     Term 19 (AT2200-0500)/CC Outputs/Current setpoint value Ch.22 <-> Data Pointer/CurrentSetpointValues[21]
//     Term 19 (AT2200-0500)/CC Outputs/Current setpoint value Ch.23 <-> Data Pointer/CurrentSetpointValues[22]
//     Term 19 (AT2200-0500)/CC Outputs/Current setpoint value Ch.24 <-> Data Pointer/CurrentSetpointValues[23]
//     Term 19 (AT2200-0500)/CC Outputs/Current setpoint value Ch.25 <-> Data Pointer/CurrentSetpointValues[24]
//     Term 19 (AT2200-0500)/CC Outputs/Current setpoint value Ch.26 <-> Data Pointer/CurrentSetpointValues[25]
//     Term 19 (AT2200-0500)/CC Outputs/Current setpoint value Ch.27 <-> Data Pointer/CurrentSetpointValues[26]
//     Term 19 (AT2200-0500)/CC Outputs/Current setpoint value Ch.28 <-> Data Pointer/CurrentSetpointValues[27]
//     Term 19 (AT2200-0500)/CC Outputs/Current setpoint value Ch.29 <-> Data Pointer/CurrentSetpointValues[28]
//     Term 19 (AT2200-0500)/CC Outputs/Current setpoint value Ch.3 <-> Data Pointer/CurrentSetpointValues[2]
//     Term 19 (AT2200-0500)/CC Outputs/Current setpoint value Ch.30 <-> Data Pointer/CurrentSetpointValues[29]
//     Term 19 (AT2200-0500)/CC Outputs/Current setpoint value Ch.4 <-> Data Pointer/CurrentSetpointValues[3]
//     Term 19 (AT2200-0500)/CC Outputs/Current setpoint value Ch.5 <-> Data Pointer/CurrentSetpointValues[4]
//     Term 19 (AT2200-0500)/CC Outputs/Current setpoint value Ch.6 <-> Data Pointer/CurrentSetpointValues[5]
//     Term 19 (AT2200-0500)/CC Outputs/Current setpoint value Ch.7 <-> Data Pointer/CurrentSetpointValues[6]
